// eDataMappingVarNames.peakshavebox_Powermonitor_ar_ApparentPower_L1: 				st_Variable:= IotExtractType(monitor.peakshavebox.Powermonitor.ar_ApparentPower[1], 1, 1); 
// eDataMappingVarNames.peakshavebox_Powermonitor_ar_ApparentPower_L2: 				st_Variable:= IotExtractType(monitor.peakshavebox.Powermonitor.ar_ApparentPower[2], 1, 1); 
// eDataMappingVarNames.peakshavebox_Powermonitor_ar_ApparentPower_L3: 				st_Variable:= IotExtractType(monitor.peakshavebox.Powermonitor.ar_ApparentPower[3], 1, 1); 
// eDataMappingVarNames.peakshavebox_Powermonitor_ar_ReactivePower_AVG: 				st_Variable:= IotExtractType(monitor.peakshavebox.Powermonitor.ar_ReactivePower[0], 1, 1); 
// eDataMappingVarNames.peakshavebox_Powermonitor_ar_ReactivePower_L1: 				st_Variable:= IotExtractType(monitor.peakshavebox.Powermonitor.ar_ReactivePower[1], 1, 1); 
// eDataMappingVarNames.peakshavebox_Powermonitor_ar_ReactivePower_L2: 				st_Variable:= IotExtractType(monitor.peakshavebox.Powermonitor.ar_ReactivePower[2], 1, 1); 
// eDataMappingVarNames.peakshavebox_Powermonitor_ar_ReactivePower_L3: 				st_Variable:= IotExtractType(monitor.peakshavebox.Powermonitor.ar_ReactivePower[3], 1, 1); 
// eDataMappingVarNames.peakshavebox_Powermonitor_ar_ActivePower_AVG: 				st_Variable:= IotExtractType(monitor.peakshavebox.Powermonitor.ar_ActivePower[0], 1, 1); 
// eDataMappingVarNames.peakshavebox_Powermonitor_ar_ActivePower_L1: 				st_Variable:= IotExtractType(monitor.peakshavebox.Powermonitor.ar_ActivePower[1], 1, 1); 
// eDataMappingVarNames.peakshavebox_Powermonitor_ar_ActivePower_L2: 				st_Variable:= IotExtractType(monitor.peakshavebox.Powermonitor.ar_ActivePower[2], 1, 1); 
// eDataMappingVarNames.peakshavebox_Powermonitor_ar_ActivePower_L3: 				st_Variable:= IotExtractType(monitor.peakshavebox.Powermonitor.ar_ActivePower[3], 1, 1); 
// eDataMappingVarNames.peakshavebox_Powermonitor_r_EnergyConsumed: 				st_Variable:= IotExtractType(monitor.peakshavebox.Powermonitor.r_EnergyConsumed, 0, 0); 
// eDataMappingVarNames.peakshavebox_Powermonitor_r_EnergySupplied: 				st_Variable:= IotExtractType(monitor.peakshavebox.Powermonitor.r_EnergySupplied, 0, 0); 
// eDataMappingVarNames.peakshavebox_Powermonitor_ar_THD_AVG: 				st_Variable:= IotExtractType(monitor.peakshavebox.Powermonitor.ar_THD[0], 1, 0); 
// eDataMappingVarNames.peakshavebox_Powermonitor_ar_THD_L1: 				st_Variable:= IotExtractType(monitor.peakshavebox.Powermonitor.ar_THD[1], 1, 0); 
// eDataMappingVarNames.peakshavebox_Powermonitor_ar_THD_L2: 				st_Variable:= IotExtractType(monitor.peakshavebox.Powermonitor.ar_THD[2], 1, 0); 
// eDataMappingVarNames.peakshavebox_Powermonitor_ar_THD_L3: 				st_Variable:= IotExtractType(monitor.peakshavebox.Powermonitor.ar_THD[3], 1, 0); 
// eDataMappingVarNames.peakshavebox_Powermonitor_ar_PowerFactor_AVG: 				st_Variable:= IotExtractType(monitor.peakshavebox.Powermonitor.ar_PowerFactor[0], 2, 0); 
// eDataMappingVarNames.peakshavebox_Powermonitor_ar_PowerFactor_L1: 				st_Variable:= IotExtractType(monitor.peakshavebox.Powermonitor.ar_PowerFactor[1], 2, 0); 
// eDataMappingVarNames.peakshavebox_Powermonitor_ar_PowerFactor_L2: 				st_Variable:= IotExtractType(monitor.peakshavebox.Powermonitor.ar_PowerFactor[2], 2, 0); 
// eDataMappingVarNames.peakshavebox_Powermonitor_ar_PowerFactor_L3: 				st_Variable:= IotExtractType(monitor.peakshavebox.Powermonitor.ar_PowerFactor[3], 2, 0); 
// eDataMappingVarNames.peakshavebox_Powermonitor_ar_Current_AVG: 				st_Variable:= IotExtractType(monitor.peakshavebox.Powermonitor.ar_Current[0], 1, 1); 
// eDataMappingVarNames.peakshavebox_Powermonitor_ar_Current_L1: 				st_Variable:= IotExtractType(monitor.peakshavebox.Powermonitor.ar_Current[1], 1, 1); 
// eDataMappingVarNames.peakshavebox_Powermonitor_ar_Current_L2: 				st_Variable:= IotExtractType(monitor.peakshavebox.Powermonitor.ar_Current[2], 1, 1); 
// eDataMappingVarNames.peakshavebox_Powermonitor_ar_Current_L3: 				st_Variable:= IotExtractType(monitor.peakshavebox.Powermonitor.ar_Current[3], 1, 1); 
// eDataMappingVarNames.peakshavebox_Powermonitor_ar_Current_N: 				st_Variable:= IotExtractType(monitor.peakshavebox.Powermonitor.ar_Current[4], 1, 1); 
// eDataMappingVarNames.peakshavebox_Powermonitor_r_CurrentUnbalance: 				st_Variable:= IotExtractType(monitor.peakshavebox.Powermonitor.r_CurrentUnbalance, 1, 0); 
// eDataMappingVarNames.peakshavebox_Powermonitor_e_ACrotationStatus: 				st_Variable:= IotExtractType(monitor.peakshavebox.Powermonitor.e_ACrotationStatus, 0, 0); 
// eDataMappingVarNames.peakshavebox_Powermonitor_ar_PhaseVoltage_AVG: 				st_Variable:= IotExtractType(monitor.peakshavebox.Powermonitor.ar_PhaseVoltage[0], 0, 0); 
// eDataMappingVarNames.peakshavebox_Powermonitor_ar_PhaseVoltage_L1: 				st_Variable:= IotExtractType(monitor.peakshavebox.Powermonitor.ar_PhaseVoltage[1], 1, 1); 
// eDataMappingVarNames.peakshavebox_Powermonitor_ar_PhaseVoltage_L2: 				st_Variable:= IotExtractType(monitor.peakshavebox.Powermonitor.ar_PhaseVoltage[2], 1, 1); 
// eDataMappingVarNames.peakshavebox_Powermonitor_ar_PhaseVoltage_L3: 				st_Variable:= IotExtractType(monitor.peakshavebox.Powermonitor.ar_PhaseVoltage[3], 1, 1); 
// eDataMappingVarNames.peakshavebox_Powermonitor_ar_LineVoltage_AVG: 				st_Variable:= IotExtractType(monitor.peakshavebox.Powermonitor.ar_LineVoltage[0], 1, 1); 
// eDataMappingVarNames.peakshavebox_Powermonitor_ar_LineVoltage_L1: 				st_Variable:= IotExtractType(monitor.peakshavebox.Powermonitor.ar_LineVoltage[1], 1, 1); 
// eDataMappingVarNames.peakshavebox_Powermonitor_ar_LineVoltage_L2: 				st_Variable:= IotExtractType(monitor.peakshavebox.Powermonitor.ar_LineVoltage[2], 1, 1); 
// eDataMappingVarNames.peakshavebox_Powermonitor_ar_LineVoltage_L3: 				st_Variable:= IotExtractType(monitor.peakshavebox.Powermonitor.ar_LineVoltage[3], 1, 1); 
// eDataMappingVarNames.peakshavebox_Powermonitor_li_TimeVoltZeroCrossup: 				st_Variable:= IotExtractType(monitor.peakshavebox.Powermonitor.li_TimeVoltZeroCrossup, 0, 0); 
// eDataMappingVarNames.peakshavebox_Powermonitor_ar_Frequency_AVG: 				st_Variable:= IotExtractType(monitor.peakshavebox.Powermonitor.ar_Frequency[0], 2, 1); 
// eDataMappingVarNames.peakshavebox_Powermonitor_ar_Frequency_L1: 				st_Variable:= IotExtractType(monitor.peakshavebox.Powermonitor.ar_Frequency[1], 2, 1); 
// eDataMappingVarNames.peakshavebox_Powermonitor_ar_Frequency_L2: 				st_Variable:= IotExtractType(monitor.peakshavebox.Powermonitor.ar_Frequency[2], 2, 1); 
// eDataMappingVarNames.peakshavebox_Powermonitor_ar_Frequency_L3: 				st_Variable:= IotExtractType(monitor.peakshavebox.Powermonitor.ar_Frequency[3], 2, 1); 
// eDataMappingVarNames.peakshavebox_Powermonitor_r_VoltageUnbalance: 				st_Variable:= IotExtractType(monitor.peakshavebox.Powermonitor.r_VoltageUnbalance, 1, 0); 
// eDataMappingVarNames.peakshavebox_PowerStatus_b_RotaryField: 				st_Variable:= IotExtractType(monitor.peakshavebox.PowerStatus.b_RotaryField, 0, 0); 
// eDataMappingVarNames.peakshavebox_PowerStatus_b_GeneralWarning: 				st_Variable:= IotExtractType(monitor.peakshavebox.PowerStatus.b_GeneralWarning, 0, 0); 
// eDataMappingVarNames.peakshavebox_PowerStatus_b_GeneralFault: 				st_Variable:= IotExtractType(monitor.peakshavebox.PowerStatus.b_GeneralFault, 0, 0); 
// eDataMappingVarNames.peakshavebox_PowerStatus_b_OverVoltage: 				st_Variable:= IotExtractType(monitor.peakshavebox.PowerStatus.b_OverVoltage, 0, 0); 
// eDataMappingVarNames.peakshavebox_PowerStatus_b_UnderVoltage: 				st_Variable:= IotExtractType(monitor.peakshavebox.PowerStatus.b_UnderVoltage, 0, 0); 
// eDataMappingVarNames.peakshavebox_PowerStatus_b_OverCurrent: 				st_Variable:= IotExtractType(monitor.peakshavebox.PowerStatus.b_OverCurrent, 0, 0); 
// eDataMappingVarNames.peakshavebox_PowerStatus_b_Error_Phase_1: 				st_Variable:= IotExtractType(monitor.peakshavebox.PowerStatus.b_Error_Phase[1], 0, 0); 
// eDataMappingVarNames.peakshavebox_PowerStatus_b_Error_Phase_2: 				st_Variable:= IotExtractType(monitor.peakshavebox.PowerStatus.b_Error_Phase[2], 0, 0); 
// eDataMappingVarNames.peakshavebox_PowerStatus_b_Error_Phase_3: 				st_Variable:= IotExtractType(monitor.peakshavebox.PowerStatus.b_Error_Phase[3], 0, 0); 
// eDataMappingVarNames.peakshavebox_r_MaxCTCurrent: 				st_Variable:= IotExtractType(monitor.peakshavebox.r_MaxCTCurrent, 0, 0); 
// eDataMappingVarNames.peakshavebox_b_buscouplerReady: 				st_Variable:= IotExtractType(monitor.peakshavebox.b_buscouplerReady, 0, 0); 
// eDataMappingVarNames.peakshavebox_b_active: 				st_Variable:= IotExtractType(monitor.peakshavebox.b_active, 0, 0); 
// eDataMappingVarNames.peakshavebox_b_dataOK: 				st_Variable:= IotExtractType(monitor.peakshavebox.b_dataOK, 0, 0); 
// eDataMappingVarNames.peakshavebox_b_ContactorFb: 				st_Variable:= IotExtractType(monitor.peakshavebox.b_ContactorFb, 0, 0); 
// eDataMappingVarNames.peakshavebox_b_SyncFb: 				st_Variable:= IotExtractType(monitor.peakshavebox.b_SyncFb, 0, 0); 
// eDataMappingVarNames.peakshavebox_b_SettingsChangePending: 				st_Variable:= IotExtractType(monitor.peakshavebox.b_SettingsChangePending, 0, 0); 
// eDataMappingVarNames.enclosure_climate_r_Humidity: 				st_Variable:= IotExtractType(monitor.enclosure.climate.r_Humidity, 1, 0); 
// eDataMappingVarNames.enclosure_climate_r_Temperature: 				st_Variable:= IotExtractType(monitor.enclosure.climate.r_Temperature, 1, 0); 
// eDataMappingVarNames.enclosure_climate_events_b_HumidityHigh: 				st_Variable:= IotExtractType(monitor.enclosure.climate.events.b_HumidityHigh, 0, 0); 
// eDataMappingVarNames.enclosure_climate_events_b_HumidityTooHigh: 				st_Variable:= IotExtractType(monitor.enclosure.climate.events.b_HumidityTooHigh, 0, 0); 
// eDataMappingVarNames.enclosure_climate_events_b_TemperatureHigh: 				st_Variable:= IotExtractType(monitor.enclosure.climate.events.b_TemperatureHigh, 0, 0); 
// eDataMappingVarNames.enclosure_climate_events_b_TemperatureTooHigh: 				st_Variable:= IotExtractType(monitor.enclosure.climate.events.b_TemperatureTooHigh, 0, 0); 
// eDataMappingVarNames.enclosure_climate_events_b_TemperatureLow: 				st_Variable:= IotExtractType(monitor.enclosure.climate.events.b_TemperatureLow, 0, 0); 
// eDataMappingVarNames.enclosure_climate_events_b_TemperatureTooLow: 				st_Variable:= IotExtractType(monitor.enclosure.climate.events.b_TemperatureTooLow, 0, 0); 
// eDataMappingVarNames.enclosure_climate_events_b_AIOverrange: 				st_Variable:= IotExtractType(monitor.enclosure.climate.events.b_AIOverrange, 0, 0); 
// eDataMappingVarNames.enclosure_climate_events_b_AIUnderrange: 				st_Variable:= IotExtractType(monitor.enclosure.climate.events.b_AIUnderrange, 0, 0); 
// eDataMappingVarNames.enclosure_climate_events_b_AIError: 				st_Variable:= IotExtractType(monitor.enclosure.climate.events.b_AIError, 0, 0); 
// eDataMappingVarNames.enclosure_climate_events_b_DewpointTooHigh: 				st_Variable:= IotExtractType(monitor.enclosure.climate.events.b_DewpointTooHigh, 0, 0); 
// //eDataMappingVarNames.enclosure_doors_b_ClientpanelDoorClosed: 				st_Variable:= IotExtractType(monitor.enclosure.doors.b_ClientpanelDoorClosed, 0, 0); 
// //eDataMappingVarNames.enclosure_doors_b_ControlPanelDoorClosed: 				st_Variable:= IotExtractType(monitor.enclosure.doors.b_ControlPanelDoorClosed, 0, 0); 
// eDataMappingVarNames.enclosure_ledstrip_b_error: 				st_Variable:= IotExtractType(monitor.enclosure.ledstrip.b_error, 0, 0); 
// eDataMappingVarNames.enclosure_ledstrip_BeckhoffLed: 				st_Variable:= IotExtractType(monitor.enclosure.ledstrip.BeckhoffLed, 0, 0); 
// eDataMappingVarNames.internalpsu_b_24VdcAvailable: 				st_Variable:= IotExtractType(monitor.internalpsu.b_24VdcAvailable, 0, 0); 
// eDataMappingVarNames.internalpsu_b_HVDCAvailable: 				st_Variable:= IotExtractType(monitor.internalpsu.b_HVDCAvailable, 0, 0); 
// eDataMappingVarNames.internalpsu_b_400VACAvailable: 				st_Variable:= IotExtractType(monitor.internalpsu.b_400VACAvailable, 0, 0); 
// //eDataMappingVarNames.internalpsu_e_400VSupplySource: 				st_Variable:= IotExtractType(monitor.internalpsu.e_400VSupplySource, 0, 0); 
// eDataMappingVarNames.internalpsu_UPS_r_InputVoltage: 				st_Variable:= IotExtractType(monitor.internalpsu.UPS.r_InputVoltage, 1, 1); 
// eDataMappingVarNames.internalpsu_UPS_r_OutputVoltage: 				st_Variable:= IotExtractType(monitor.internalpsu.UPS.r_OutputVoltage, 1, 1); 
// eDataMappingVarNames.internalpsu_UPS_r_BatteryVoltage: 				st_Variable:= IotExtractType(monitor.internalpsu.UPS.r_BatteryVoltage, 1, 1); 
// eDataMappingVarNames.internalpsu_UPS_r_OutputCurrent: 				st_Variable:= IotExtractType(monitor.internalpsu.UPS.r_OutputCurrent, 2, 0); 
// eDataMappingVarNames.internalpsu_UPS_ui_SOC: 				st_Variable:= IotExtractType(monitor.internalpsu.UPS.ui_SOC, 0, 0); 
// eDataMappingVarNames.internalpsu_UPS_b_ChargerActive: 				st_Variable:= IotExtractType(monitor.internalpsu.UPS.b_ChargerActive, 0, 0); 
// eDataMappingVarNames.internalpsu_UPS_b_SystemOnBattery: 				st_Variable:= IotExtractType(monitor.internalpsu.UPS.b_SystemOnBattery, 0, 0); 
// eDataMappingVarNames.internalpsu_UPS_b_SystemOnDCInput: 				st_Variable:= IotExtractType(monitor.internalpsu.UPS.b_SystemOnDCInput, 0, 0); 
// eDataMappingVarNames.internalpsu_UPS_Events_b_BatteryLowInfo: 				st_Variable:= IotExtractType(monitor.internalpsu.UPS.Events.b_BatteryLowInfo, 0, 0); 
// eDataMappingVarNames.internalpsu_UPS_Events_b_BatteryLowWarning: 				st_Variable:= IotExtractType(monitor.internalpsu.UPS.Events.b_BatteryLowWarning, 0, 0); 
// eDataMappingVarNames.internalpsu_UPS_Events_b_BatteryLowError: 				st_Variable:= IotExtractType(monitor.internalpsu.UPS.Events.b_BatteryLowError, 0, 0); 
// eDataMappingVarNames.internalpsu_UPS_Events_b_NoBatteryError: 				st_Variable:= IotExtractType(monitor.internalpsu.UPS.Events.b_NoBatteryError, 0, 0); 
// eDataMappingVarNames.internalpsu_UPS_Events_b_InputVoltageWarning: 				st_Variable:= IotExtractType(monitor.internalpsu.UPS.Events.b_InputVoltageWarning, 0, 0); 
// eDataMappingVarNames.internalpsu_Events_b_DCPSUFault: 				st_Variable:= IotExtractType(monitor.internalpsu.Events.b_DCPSUFault, 0, 0); 
// eDataMappingVarNames.internalpsu_Events_b_ACPSUFault: 				st_Variable:= IotExtractType(monitor.internalpsu.Events.b_ACPSUFault, 0, 0); 
// eDataMappingVarNames.internalpsu_Events_b_GridInputFuseTripped: 				st_Variable:= IotExtractType(monitor.internalpsu.Events.b_GridInputFuseTripped, 0, 0); 
// //eDataMappingVarNames.internalpsu_Events_b_CEEInputFuseTripped: 				st_Variable:= IotExtractType(monitor.internalpsu.Events.b_CEEInputFuseTripped, 0, 0); 
// eDataMappingVarNames.internalpsu_Events_b_HVDCShutdownTimeExceeded: 				st_Variable:= IotExtractType(monitor.internalpsu.Events.b_HVDCShutdownTimeExceeded, 0, 0); 
// eDataMappingVarNames.internalpsu_Events_b_UPSLowShutdown: 				st_Variable:= IotExtractType(monitor.internalpsu.Events.b_UPSLowShutdown, 0, 0); 
// eDataMappingVarNames.PLC_r_CPUload: 				st_Variable:= IotExtractType(monitor.PLC.r_CPUload, 0, 0); 
// eDataMappingVarNames.PLC_e_ProfinetState: 				st_Variable:= IotExtractType(monitor.PLC.e_ProfinetState, 0, 0); 
// eDataMappingVarNames.PLC_e_EthercatState: 				st_Variable:= IotExtractType(monitor.PLC.e_EthercatState, 0, 0); 
// eDataMappingVarNames.Cooling_CoolingSystemMode: 				st_Variable:= IotExtractType(monitor.Cooling.CoolingSystemMode, 0, 0); 
// eDataMappingVarNames.Cooling_HeatPumpStatus: 				st_Variable:= IotExtractType(monitor.Cooling.HeatPumpStatus, 0, 0); 
// eDataMappingVarNames.Cooling_r_CoolantTemperature: 				st_Variable:= IotExtractType(monitor.Cooling.r_CoolantTemperature, 1, 0); 
// eDataMappingVarNames.Cooling_r_CoolantPressure: 				st_Variable:= IotExtractType(monitor.Cooling.r_CoolantPressure, 2, 0); 
// eDataMappingVarNames.Cooling_r_EnclosureDewpoint: 				st_Variable:= IotExtractType(monitor.Cooling.r_EnclosureDewpoint, 0, 0); 
// eDataMappingVarNames.Cooling_ui_DehumRemainingTime: 				st_Variable:= IotExtractType(monitor.Cooling.ui_DehumRemainingTime, 0, 0); 
// eDataMappingVarNames.Cooling_HeatPumpSystem_HeatPumpStatus: 				st_Variable:= IotExtractType(monitor.Cooling.HeatPumpStatus, 0, 0); 
// eDataMappingVarNames.Cooling_HeatPumpSystem_PrimaryHeatpumpGet_HeatPumpState: 				st_Variable:= IotExtractType(monitor.Cooling.HeatPumpStatus, 0, 0); {warning 'needs revision, heatpump now doesn't have individuals state'} 
// eDataMappingVarNames.Cooling_HeatPumpSystem_PrimaryHeatpumpGet_Setpoint: 				st_Variable:= IotExtractType(monitor.Cooling.Heatpump.Setpoint, 0, 0); 
// eDataMappingVarNames.Cooling_HeatPumpSystem_PrimaryHeatpumpGet_Events_b_CommWarning: 				st_Variable:= IotExtractType(monitor.Cooling.Heatpump.Events.b_CommWarning, 0, 0); 
// eDataMappingVarNames.Cooling_HeatPumpSystem_PrimaryHeatpumpGet_Events_b_ProbeError: 				st_Variable:= IotExtractType(monitor.Cooling.Heatpump.Events.b_ProbeError, 0, 0); 
// eDataMappingVarNames.Cooling_HeatPumpSystem_PrimaryHeatpumpGet_Events_b_PressureError: 				st_Variable:= IotExtractType(monitor.Cooling.Heatpump.Events.b_PressureError, 0, 0); 
// eDataMappingVarNames.Cooling_HeatPumpSystem_PrimaryHeatpumpGet_Events_b_CompressorError: 				st_Variable:= IotExtractType(monitor.Cooling.Heatpump.Events.b_CompressorError, 0, 0); 
// eDataMappingVarNames.Cooling_HeatPumpSystem_PrimaryHeatpumpGet_Events_b_ValveError: 				st_Variable:= IotExtractType(monitor.Cooling.Heatpump.Events.b_ValveError, 0, 0); 
// eDataMappingVarNames.Cooling_HeatPumpSystem_PrimaryHeatpumpGet_Events_b_FanError: 				st_Variable:= IotExtractType(monitor.Cooling.Heatpump.Events.b_FanError, 0, 0); 
// eDataMappingVarNames.Cooling_HeatPumpSystem_PrimaryHeatpumpGet_Events_b_PumpError: 				st_Variable:= IotExtractType(monitor.Cooling.Heatpump.Events.b_PumpError, 0, 0); 
// eDataMappingVarNames.Cooling_HeatPumpSystem_PrimaryHeatpumpGet_Events_b_WaterTempError: 				st_Variable:= IotExtractType(monitor.Cooling.Heatpump.Events.b_WaterTempError, 0, 0); 
// eDataMappingVarNames.Cooling_HeatPumpSystem_PrimaryHeatpumpGet_Events_b_IOError: 				st_Variable:= IotExtractType(monitor.Cooling.Heatpump.Events.b_IOError, 0, 0); 
// eDataMappingVarNames.Cooling_HeatPumpSystem_PrimaryHeatpumpGet_Events_b_HeatpumpPreheatingActive: 				st_Variable:= IotExtractType(monitor.Cooling.Heatpump.Events.b_HeatpumpPreheatingActive, 0, 0); 
// eDataMappingVarNames.Cooling_HeatPumpSystem_PrimaryHeatpumpGet_Events_b_TooColdForHeatpumpHeating: 				st_Variable:= IotExtractType(monitor.Cooling.Heatpump.Events.b_TooColdForHeatpumpHeating, 0, 0); 
// eDataMappingVarNames.Cooling_HeatPumpSystem_PrimaryHeatpumpGet_HeatpumpData_i_FW_Version: 				st_Variable:= IotExtractType(monitor.Cooling.Heatpump.HeatpumpData.i_FW_Version, 0, 0); 
// eDataMappingVarNames.Cooling_HeatPumpSystem_PrimaryHeatpumpGet_HeatpumpData_i_FW_release: 				st_Variable:= IotExtractType(monitor.Cooling.Heatpump.HeatpumpData.i_FW_release, 0, 0); 
// eDataMappingVarNames.Cooling_HeatPumpSystem_PrimaryHeatpumpGet_HeatpumpData_w_FW_Subrelease: 				st_Variable:= IotExtractType(monitor.Cooling.Heatpump.HeatpumpData.HeatpumpData.w_FW_Subrelease, 0, 0); 
// eDataMappingVarNames.Cooling_HeatPumpSystem_PrimaryHeatpumpGet_HeatpumpData_w_FW_creationDate: 				st_Variable:= IotExtractType(monitor.Cooling.Heatpump.Heatpumpdata.w_FW_creationDate, 0, 0); 
// eDataMappingVarNames.Cooling_HeatPumpSystem_PrimaryHeatpumpGet_HeatpumpData_w_Serialnumber_0: 				st_Variable:= IotExtractType(monitor.Cooling.Heatpump.Heatpumpdata.w_Serialnumber[0], 0, 0); 
// eDataMappingVarNames.Cooling_HeatPumpSystem_PrimaryHeatpumpGet_HeatpumpData_w_Serialnumber_1: 				st_Variable:= IotExtractType(monitor.Cooling.Heatpump.Heatpumpdata.w_Serialnumber[1], 0, 0); 
// eDataMappingVarNames.Cooling_HeatPumpSystem_PrimaryHeatpumpGet_HeatpumpData_w_Serialnumber_2: 				st_Variable:= IotExtractType(monitor.Cooling.Heatpump.Heatpumpdata.w_Serialnumber[2], 0, 0); 
// eDataMappingVarNames.Cooling_HeatPumpSystem_PrimaryHeatpumpGet_HeatpumpData_w_Serialnumber_3: 				st_Variable:= IotExtractType(monitor.Cooling.Heatpump.Heatpumpdata.w_Serialnumber[3], 0, 0); 
// eDataMappingVarNames.Cooling_HeatPumpSystem_PrimaryHeatpumpGet_HeatpumpData_w_Serialnumber_4: 				st_Variable:= IotExtractType(monitor.Cooling.Heatpump.Heatpumpdata.w_Serialnumber[4], 0, 0); 
// eDataMappingVarNames.Cooling_HeatPumpSystem_PrimaryHeatpumpGet_HeatpumpData_w_Serialnumber_5: 				st_Variable:= IotExtractType(monitor.Cooling.Heatpump.Heatpumpdata.w_Serialnumber[5], 0, 0); 
// eDataMappingVarNames.Cooling_HeatPumpSystem_PrimaryHeatpumpGet_HeatpumpData_w_Serialnumber_6: 				st_Variable:= IotExtractType(monitor.Cooling.Heatpump.Heatpumpdata.w_Serialnumber[6], 0, 0); 
// eDataMappingVarNames.Cooling_HeatPumpSystem_PrimaryHeatpumpGet_HeatpumpData_w_Serialnumber_7: 				st_Variable:= IotExtractType(monitor.Cooling.Heatpump.Heatpumpdata.w_Serialnumber[7], 0, 0); 
// eDataMappingVarNames.Cooling_HeatPumpSystem_PrimaryHeatpumpGet_HeatpumpData_w_Serialnumber_8: 				st_Variable:= IotExtractType(monitor.Cooling.Heatpump.Heatpumpdata.w_Serialnumber[8], 0, 0); 
// eDataMappingVarNames.Cooling_HeatPumpSystem_PrimaryHeatpumpGet_HeatpumpData_w_Serialnumber_9: 				st_Variable:= IotExtractType(monitor.Cooling.Heatpump.Heatpumpdata.w_Serialnumber[9], 0, 0); 
// eDataMappingVarNames.Cooling_HeatPumpSystem_PrimaryHeatpumpGet_HeatpumpData_w_Serialnumber_10: 				st_Variable:= IotExtractType(monitor.Cooling.Heatpump.Heatpumpdata.w_Serialnumber[10], 0, 0); 
// eDataMappingVarNames.Cooling_HeatPumpSystem_PrimaryHeatpumpGet_HeatpumpData_w_Serialnumber_11: 				st_Variable:= IotExtractType(monitor.Cooling.Heatpump.Heatpumpdata.w_Serialnumber[11], 0, 0); 
// eDataMappingVarNames.Cooling_HeatPumpSystem_PrimaryHeatpumpGet_HeatpumpData_w_Serialnumber_12: 				st_Variable:= IotExtractType(monitor.Cooling.Heatpump.Heatpumpdata.w_Serialnumber[12], 0, 0); 
// eDataMappingVarNames.Cooling_HeatPumpSystem_PrimaryHeatpumpGet_HeatpumpData_w_Serialnumber_13: 				st_Variable:= IotExtractType(monitor.Cooling.Heatpump.Heatpumpdata.w_Serialnumber[13], 0, 0); 
// eDataMappingVarNames.Cooling_HeatPumpSystem_PrimaryHeatpumpGet_HeatpumpData_w_Serialnumber_14: 				st_Variable:= IotExtractType(monitor.Cooling.Heatpump.Heatpumpdata.w_Serialnumber[14], 0, 0); 
// eDataMappingVarNames.Cooling_HeatPumpSystem_PrimaryHeatpumpGet_HeatpumpData_w_Serialnumber_15: 				st_Variable:= IotExtractType(monitor.Cooling.Heatpump.Heatpumpdata.w_Serialnumber[15], 0, 0); 
// eDataMappingVarNames.Cooling_HeatPumpSystem_PrimaryHeatpumpGet_HeatpumpData_w_Serialnumber_16: 				st_Variable:= IotExtractType(monitor.Cooling.Heatpump.Heatpumpdata.w_Serialnumber[16], 0, 0); 
// eDataMappingVarNames.Cooling_HeatPumpSystem_PrimaryHeatpumpGet_HeatpumpData_w_Serialnumber_17: 				st_Variable:= IotExtractType(monitor.Cooling.Heatpump.Heatpumpdata.w_Serialnumber[17], 0, 0); 
// eDataMappingVarNames.Cooling_HeatPumpSystem_PrimaryHeatpumpGet_HeatpumpData_i_OperatingHours: 				st_Variable:= IotExtractType(monitor.Cooling.Heatpump.Heatpumpdata.i_OperatingHours, 0, 0); 
// eDataMappingVarNames.Cooling_HeatPumpSystem_PrimaryHeatpumpGet_HeatpumpData_r_CoolantPower: 				st_Variable:= IotExtractType(monitor.Cooling.Heatpump.Heatpumpdata.r_CoolantPower, 0, 0); 
// eDataMappingVarNames.Cooling_HeatPumpSystem_PrimaryHeatpumpGet_HeatpumpData_r_InletWaterTemp: 				st_Variable:= IotExtractType(monitor.Cooling.Heatpump.Heatpumpdata.r_InletWaterTemp, 0, 0); 
// eDataMappingVarNames.Cooling_HeatPumpSystem_PrimaryHeatpumpGet_HeatpumpData_r_OutletWaterTemp: 				st_Variable:= IotExtractType(monitor.Cooling.Heatpump.Heatpumpdata.r_OutletWaterTemp, 0, 0); 
// eDataMappingVarNames.Cooling_HeatPumpSystem_PrimaryHeatpumpGet_HeatpumpData_r_HighPressure: 				st_Variable:= IotExtractType(monitor.Cooling.Heatpump.Heatpumpdata.r_HighPressure, 0, 0); 
// eDataMappingVarNames.Cooling_HeatPumpSystem_PrimaryHeatpumpGet_HeatpumpData_r_LowPressure: 				st_Variable:= IotExtractType(monitor.Cooling.HeatPump.HeatpumpData.r_LowPressure, 0, 0); 
// eDataMappingVarNames.Cooling_HeatPumpSystem_PrimaryHeatpumpGet_HeatpumpData_r_CompInputTemp: 				st_Variable:= IotExtractType(monitor.Cooling.Heatpump.HeatpumpData.r_CompInputTemp, 0, 0); 
// eDataMappingVarNames.Cooling_HeatPumpSystem_PrimaryHeatpumpGet_HeatpumpData_r_OutdoorTemp: 				st_Variable:= IotExtractType(monitor.Cooling.Heatpump.HeatpumpData.r_OutdoorTemp, 0, 0); 
// eDataMappingVarNames.Cooling_HeatPumpSystem_PrimaryHeatpumpGet_HeatpumpData_r_CompOutputTemp: 				st_Variable:= IotExtractType(monitor.Cooling.Heatpump.HeatpumpData.r_CompOutputTemp, 0, 0); 
// eDataMappingVarNames.Cooling_HeatPumpSystem_PrimaryHeatpumpGet_HeatpumpData_ui_WaterFlowRate: 				st_Variable:= IotExtractType(monitor.Cooling.Heatpump.HeatpumpData.ui_WaterFlowRate, 0, 0); 
// eDataMappingVarNames.Cooling_HeatPumpSystem_PrimaryHeatpumpGet_HeatpumpData_w_ErrorList_1: 				st_Variable:= IotExtractType(monitor.Cooling.Heatpump.HeatpumpData.w_ErrorList[1], 0, 0); 
// eDataMappingVarNames.Cooling_HeatPumpSystem_PrimaryHeatpumpGet_HeatpumpData_w_ErrorList_2: 				st_Variable:= IotExtractType(monitor.Cooling.Heatpump.HeatpumpData.w_ErrorList[2], 0, 0); 
// eDataMappingVarNames.Cooling_HeatPumpSystem_PrimaryHeatpumpGet_HeatpumpData_w_ErrorList_3: 				st_Variable:= IotExtractType(monitor.Cooling.Heatpump.HeatpumpData.w_ErrorList[3], 0, 0); 
// eDataMappingVarNames.Cooling_HeatPumpSystem_PrimaryHeatpumpGet_HeatpumpData_w_ErrorList_4: 				st_Variable:= IotExtractType(monitor.Cooling.Heatpump.HeatpumpData.w_ErrorList[4], 0, 0); 
// eDataMappingVarNames.Cooling_HeatPumpSystem_PrimaryHeatpumpGet_HeatpumpData_w_ErrorList_5: 				st_Variable:= IotExtractType(monitor.Cooling.Heatpump.HeatpumpData.w_ErrorList[5], 0, 0); 
// eDataMappingVarNames.Cooling_HeatPumpSystem_PrimaryHeatpumpGet_HeatpumpData_w_ErrorList_6: 				st_Variable:= IotExtractType(monitor.Cooling.Heatpump.HeatpumpData.w_ErrorList[6], 0, 0); 
// eDataMappingVarNames.Cooling_HeatPumpSystem_PrimaryHeatpumpGet_HeatpumpData_w_ErrorList_7: 				st_Variable:= IotExtractType(monitor.Cooling.Heatpump.HeatpumpData.w_ErrorList[7], 0, 0); 
// eDataMappingVarNames.Cooling_HeatPumpSystem_PrimaryHeatpumpGet_HeatpumpData_r_FanSpeedPCT: 				st_Variable:= IotExtractType(monitor.Cooling.Heatpump.HeatpumpData.r_FanSpeedPCT, 0, 0); 
// eDataMappingVarNames.Cooling_HeatPumpSystem_PrimaryHeatpumpGet_HeatpumpData_r_PumpSpeedPCT: 				st_Variable:= IotExtractType(monitor.Cooling.Heatpump.HeatpumpData.r_PumpSpeedPCT, 0, 0); 
// eDataMappingVarNames.Cooling_HeatPumpSystem_PrimaryHeatpumpGet_HeatpumpData_r_SetpointHeating: 				st_Variable:= IotExtractType(monitor.Cooling.Heatpump.HeatpumpData.r_SetpointHeating, 1, 0); 
// eDataMappingVarNames.Cooling_HeatPumpSystem_PrimaryHeatpumpGet_HeatpumpData_r_SetpointCooling: 				st_Variable:= IotExtractType(monitor.Cooling.Heatpump.HeatpumpData.r_SetpointCooling, 1, 0); 
// eDataMappingVarNames.Cooling_HeatPumpSystem_PrimaryHeatpumpGet_HeatpumpData_b_DefrostingActive: 				st_Variable:= IotExtractType(monitor.Cooling.Heatpump.HeatpumpData.b_DefrostingActive, 0, 0); 
// eDataMappingVarNames.Cooling_HeatPumpSystem_SecondaryHeatpumpGet_HeatPumpState: 				st_Variable:= IotExtractType(monitor.Cooling.HeatPumpSystem.SecondaryHeatpumpGet.HeatPumpState, 0, 0); 
// eDataMappingVarNames.Cooling_HeatPumpSystem_SecondaryHeatpumpGet_Setpoint: 				st_Variable:= IotExtractType(monitor.Cooling.HeatPumpSystem.SecondaryHeatpumpGet.Setpoint, 0, 0); 
// eDataMappingVarNames.Cooling_HeatPumpSystem_SecondaryHeatpumpGet_Events_b_CommWarning: 				st_Variable:= IotExtractType(monitor.Cooling.HeatPumpSystem.SecondaryHeatpumpGet.Events.b_CommWarning, 0, 0); 
// eDataMappingVarNames.Cooling_HeatPumpSystem_SecondaryHeatpumpGet_Events_b_ProbeError: 				st_Variable:= IotExtractType(monitor.Cooling.HeatPumpSystem.SecondaryHeatpumpGet.Events.b_ProbeError, 0, 0); 
// eDataMappingVarNames.Cooling_HeatPumpSystem_SecondaryHeatpumpGet_Events_b_PressureError: 				st_Variable:= IotExtractType(monitor.Cooling.HeatPumpSystem.SecondaryHeatpumpGet.Events.b_PressureError, 0, 0); 
// eDataMappingVarNames.Cooling_HeatPumpSystem_SecondaryHeatpumpGet_Events_b_CompressorError: 				st_Variable:= IotExtractType(monitor.Cooling.HeatPumpSystem.SecondaryHeatpumpGet.Events.b_CompressorError, 0, 0); 
// eDataMappingVarNames.Cooling_HeatPumpSystem_SecondaryHeatpumpGet_Events_b_ValveError: 				st_Variable:= IotExtractType(monitor.Cooling.HeatPumpSystem.SecondaryHeatpumpGet.Events.b_ValveError, 0, 0); 
// eDataMappingVarNames.Cooling_HeatPumpSystem_SecondaryHeatpumpGet_Events_b_FanError: 				st_Variable:= IotExtractType(monitor.Cooling.HeatPumpSystem.SecondaryHeatpumpGet.Events.b_FanError, 0, 0); 
// eDataMappingVarNames.Cooling_HeatPumpSystem_SecondaryHeatpumpGet_Events_b_PumpError: 				st_Variable:= IotExtractType(monitor.Cooling.HeatPumpSystem.SecondaryHeatpumpGet.Events.b_PumpError, 0, 0); 
// eDataMappingVarNames.Cooling_HeatPumpSystem_SecondaryHeatpumpGet_Events_b_WaterTempError: 				st_Variable:= IotExtractType(monitor.Cooling.HeatPumpSystem.SecondaryHeatpumpGet.Events.b_WaterTempError, 0, 0); 
// eDataMappingVarNames.Cooling_HeatPumpSystem_SecondaryHeatpumpGet_Events_b_IOError: 				st_Variable:= IotExtractType(monitor.Cooling.HeatPumpSystem.SecondaryHeatpumpGet.Events.b_IOError, 0, 0); 
// eDataMappingVarNames.Cooling_HeatPumpSystem_SecondaryHeatpumpGet_Events_b_HeatpumpPreheatingActive: 				st_Variable:= IotExtractType(monitor.Cooling.HeatPumpSystem.SecondaryHeatpumpGet.Events.b_HeatpumpPreheatingActive, 0, 0); 
// eDataMappingVarNames.Cooling_HeatPumpSystem_SecondaryHeatpumpGet_Events_b_TooColdForHeatpumpHeating: 				st_Variable:= IotExtractType(monitor.Cooling.HeatPumpSystem.SecondaryHeatpumpGet.Events.b_TooColdForHeatpumpHeating, 0, 0); 
// eDataMappingVarNames.Cooling_HeatPumpSystem_SecondaryHeatpumpGet_HeatpumpData_i_FW_Version: 				st_Variable:= IotExtractType(monitor.Cooling.HeatPumpSystem.SecondaryHeatpumpGet.HeatpumpData.i_FW_Version, 0, 0); 
// eDataMappingVarNames.Cooling_HeatPumpSystem_SecondaryHeatpumpGet_HeatpumpData_i_FW_release: 				st_Variable:= IotExtractType(monitor.Cooling.HeatPumpSystem.SecondaryHeatpumpGet.HeatpumpData.i_FW_release, 0, 0); 
// eDataMappingVarNames.Cooling_HeatPumpSystem_SecondaryHeatpumpGet_HeatpumpData_w_FW_Subrelease: 				st_Variable:= IotExtractType(monitor.Cooling.HeatPumpSystem.SecondaryHeatpumpGet.HeatpumpData.w_FW_Subrelease, 0, 0); 
// eDataMappingVarNames.Cooling_HeatPumpSystem_SecondaryHeatpumpGet_HeatpumpData_w_FW_creationDate: 				st_Variable:= IotExtractType(monitor.Cooling.HeatPumpSystem.SecondaryHeatpumpGet.HeatpumpData.w_FW_creationDate, 0, 0); 
// eDataMappingVarNames.Cooling_HeatPumpSystem_SecondaryHeatpumpGet_HeatpumpData_w_Serialnumber_0: 				st_Variable:= IotExtractType(monitor.Cooling.HeatPumpSystem.SecondaryHeatpumpGet.HeatpumpData.w_Serialnumber[0], 0, 0); 
// eDataMappingVarNames.Cooling_HeatPumpSystem_SecondaryHeatpumpGet_HeatpumpData_w_Serialnumber_1: 				st_Variable:= IotExtractType(monitor.Cooling.HeatPumpSystem.SecondaryHeatpumpGet.HeatpumpData.w_Serialnumber[1], 0, 0); 
// eDataMappingVarNames.Cooling_HeatPumpSystem_SecondaryHeatpumpGet_HeatpumpData_w_Serialnumber_2: 				st_Variable:= IotExtractType(monitor.Cooling.HeatPumpSystem.SecondaryHeatpumpGet.HeatpumpData.w_Serialnumber[2], 0, 0); 
// eDataMappingVarNames.Cooling_HeatPumpSystem_SecondaryHeatpumpGet_HeatpumpData_w_Serialnumber_3: 				st_Variable:= IotExtractType(monitor.Cooling.HeatPumpSystem.SecondaryHeatpumpGet.HeatpumpData.w_Serialnumber[3], 0, 0); 
// eDataMappingVarNames.Cooling_HeatPumpSystem_SecondaryHeatpumpGet_HeatpumpData_w_Serialnumber_4: 				st_Variable:= IotExtractType(monitor.Cooling.HeatPumpSystem.SecondaryHeatpumpGet.HeatpumpData.w_Serialnumber[4], 0, 0); 
// eDataMappingVarNames.Cooling_HeatPumpSystem_SecondaryHeatpumpGet_HeatpumpData_w_Serialnumber_5: 				st_Variable:= IotExtractType(monitor.Cooling.HeatPumpSystem.SecondaryHeatpumpGet.HeatpumpData.w_Serialnumber[5], 0, 0); 
// eDataMappingVarNames.Cooling_HeatPumpSystem_SecondaryHeatpumpGet_HeatpumpData_w_Serialnumber_6: 				st_Variable:= IotExtractType(monitor.Cooling.HeatPumpSystem.SecondaryHeatpumpGet.HeatpumpData.w_Serialnumber[6], 0, 0); 
// eDataMappingVarNames.Cooling_HeatPumpSystem_SecondaryHeatpumpGet_HeatpumpData_w_Serialnumber_7: 				st_Variable:= IotExtractType(monitor.Cooling.HeatPumpSystem.SecondaryHeatpumpGet.HeatpumpData.w_Serialnumber[7], 0, 0); 
// eDataMappingVarNames.Cooling_HeatPumpSystem_SecondaryHeatpumpGet_HeatpumpData_w_Serialnumber_8: 				st_Variable:= IotExtractType(monitor.Cooling.HeatPumpSystem.SecondaryHeatpumpGet.HeatpumpData.w_Serialnumber[8], 0, 0); 
// eDataMappingVarNames.Cooling_HeatPumpSystem_SecondaryHeatpumpGet_HeatpumpData_w_Serialnumber_9: 				st_Variable:= IotExtractType(monitor.Cooling.HeatPumpSystem.SecondaryHeatpumpGet.HeatpumpData.w_Serialnumber[9], 0, 0); 
// eDataMappingVarNames.Cooling_HeatPumpSystem_SecondaryHeatpumpGet_HeatpumpData_w_Serialnumber_10: 				st_Variable:= IotExtractType(monitor.Cooling.HeatPumpSystem.SecondaryHeatpumpGet.HeatpumpData.w_Serialnumber[10], 0, 0); 
// eDataMappingVarNames.Cooling_HeatPumpSystem_SecondaryHeatpumpGet_HeatpumpData_w_Serialnumber_11: 				st_Variable:= IotExtractType(monitor.Cooling.HeatPumpSystem.SecondaryHeatpumpGet.HeatpumpData.w_Serialnumber[11], 0, 0); 
// eDataMappingVarNames.Cooling_HeatPumpSystem_SecondaryHeatpumpGet_HeatpumpData_w_Serialnumber_12: 				st_Variable:= IotExtractType(monitor.Cooling.HeatPumpSystem.SecondaryHeatpumpGet.HeatpumpData.w_Serialnumber[12], 0, 0); 
// eDataMappingVarNames.Cooling_HeatPumpSystem_SecondaryHeatpumpGet_HeatpumpData_w_Serialnumber_13: 				st_Variable:= IotExtractType(monitor.Cooling.HeatPumpSystem.SecondaryHeatpumpGet.HeatpumpData.w_Serialnumber[13], 0, 0); 
// eDataMappingVarNames.Cooling_HeatPumpSystem_SecondaryHeatpumpGet_HeatpumpData_w_Serialnumber_14: 				st_Variable:= IotExtractType(monitor.Cooling.HeatPumpSystem.SecondaryHeatpumpGet.HeatpumpData.w_Serialnumber[14], 0, 0); 
// eDataMappingVarNames.Cooling_HeatPumpSystem_SecondaryHeatpumpGet_HeatpumpData_w_Serialnumber_15: 				st_Variable:= IotExtractType(monitor.Cooling.HeatPumpSystem.SecondaryHeatpumpGet.HeatpumpData.w_Serialnumber[15], 0, 0); 
// eDataMappingVarNames.Cooling_HeatPumpSystem_SecondaryHeatpumpGet_HeatpumpData_w_Serialnumber_16: 				st_Variable:= IotExtractType(monitor.Cooling.HeatPumpSystem.SecondaryHeatpumpGet.HeatpumpData.w_Serialnumber[16], 0, 0); 
// eDataMappingVarNames.Cooling_HeatPumpSystem_SecondaryHeatpumpGet_HeatpumpData_w_Serialnumber_17: 				st_Variable:= IotExtractType(monitor.Cooling.HeatPumpSystem.SecondaryHeatpumpGet.HeatpumpData.w_Serialnumber[17], 0, 0); 
// eDataMappingVarNames.Cooling_HeatPumpSystem_SecondaryHeatpumpGet_HeatpumpData_i_OperatingHours: 				st_Variable:= IotExtractType(monitor.Cooling.HeatPumpSystem.SecondaryHeatpumpGet.HeatpumpData.i_OperatingHours, 0, 0); 
// eDataMappingVarNames.Cooling_HeatPumpSystem_SecondaryHeatpumpGet_HeatpumpData_r_CoolantPower: 				st_Variable:= IotExtractType(monitor.Cooling.HeatPumpSystem.SecondaryHeatpumpGet.HeatpumpData.r_CoolantPower, 1, 0); 
// eDataMappingVarNames.Cooling_HeatPumpSystem_SecondaryHeatpumpGet_HeatpumpData_r_InletWaterTemp: 				st_Variable:= IotExtractType(monitor.Cooling.HeatPumpSystem.SecondaryHeatpumpGet.HeatpumpData.r_InletWaterTemp, 1, 0); 
// eDataMappingVarNames.Cooling_HeatPumpSystem_SecondaryHeatpumpGet_HeatpumpData_r_OutletWaterTemp: 				st_Variable:= IotExtractType(monitor.Cooling.HeatPumpSystem.SecondaryHeatpumpGet.HeatpumpData.r_OutletWaterTemp, 1, 0); 
// eDataMappingVarNames.Cooling_HeatPumpSystem_SecondaryHeatpumpGet_HeatpumpData_r_HighPressure: 				st_Variable:= IotExtractType(monitor.Cooling.HeatPumpSystem.SecondaryHeatpumpGet.HeatpumpData.r_HighPressure, 1, 0); 
// eDataMappingVarNames.Cooling_HeatPumpSystem_SecondaryHeatpumpGet_HeatpumpData_r_LowPressure: 				st_Variable:= IotExtractType(monitor.Cooling.HeatPumpSystem.SecondaryHeatpumpGet.HeatpumpData.r_LowPressure, 1, 0); 
// eDataMappingVarNames.Cooling_HeatPumpSystem_SecondaryHeatpumpGet_HeatpumpData_r_CompInputTemp: 				st_Variable:= IotExtractType(monitor.Cooling.HeatPumpSystem.SecondaryHeatpumpGet.HeatpumpData.r_CompInputTemp, 1, 0); 
// eDataMappingVarNames.Cooling_HeatPumpSystem_SecondaryHeatpumpGet_HeatpumpData_r_OutdoorTemp: 				st_Variable:= IotExtractType(monitor.Cooling.HeatPumpSystem.SecondaryHeatpumpGet.HeatpumpData.r_OutdoorTemp, 1, 0); 
// eDataMappingVarNames.Cooling_HeatPumpSystem_SecondaryHeatpumpGet_HeatpumpData_r_CompOutputTemp: 				st_Variable:= IotExtractType(monitor.Cooling.HeatPumpSystem.SecondaryHeatpumpGet.HeatpumpData.r_CompOutputTemp, 1, 0); 
// eDataMappingVarNames.Cooling_HeatPumpSystem_SecondaryHeatpumpGet_HeatpumpData_ui_WaterFlowRate: 				st_Variable:= IotExtractType(monitor.Cooling.HeatPumpSystem.SecondaryHeatpumpGet.HeatpumpData.ui_WaterFlowRate, 1, 0); 
// eDataMappingVarNames.Cooling_HeatPumpSystem_SecondaryHeatpumpGet_HeatpumpData_w_ErrorList_1: 				st_Variable:= IotExtractType(monitor.Cooling.HeatPumpSystem.SecondaryHeatpumpGet.HeatpumpData.w_ErrorList[1], 0, 0); 
// eDataMappingVarNames.Cooling_HeatPumpSystem_SecondaryHeatpumpGet_HeatpumpData_w_ErrorList_2: 				st_Variable:= IotExtractType(monitor.Cooling.HeatPumpSystem.SecondaryHeatpumpGet.HeatpumpData.w_ErrorList[2], 0, 0); 
// eDataMappingVarNames.Cooling_HeatPumpSystem_SecondaryHeatpumpGet_HeatpumpData_w_ErrorList_3: 				st_Variable:= IotExtractType(monitor.Cooling.HeatPumpSystem.SecondaryHeatpumpGet.HeatpumpData.w_ErrorList[3], 0, 0); 
// eDataMappingVarNames.Cooling_HeatPumpSystem_SecondaryHeatpumpGet_HeatpumpData_w_ErrorList_4: 				st_Variable:= IotExtractType(monitor.Cooling.HeatPumpSystem.SecondaryHeatpumpGet.HeatpumpData.w_ErrorList[4], 0, 0); 
// eDataMappingVarNames.Cooling_HeatPumpSystem_SecondaryHeatpumpGet_HeatpumpData_w_ErrorList_5: 				st_Variable:= IotExtractType(monitor.Cooling.HeatPumpSystem.SecondaryHeatpumpGet.HeatpumpData.w_ErrorList[5], 0, 0); 
// eDataMappingVarNames.Cooling_HeatPumpSystem_SecondaryHeatpumpGet_HeatpumpData_w_ErrorList_6: 				st_Variable:= IotExtractType(monitor.Cooling.HeatPumpSystem.SecondaryHeatpumpGet.HeatpumpData.w_ErrorList[6], 0, 0); 
// eDataMappingVarNames.Cooling_HeatPumpSystem_SecondaryHeatpumpGet_HeatpumpData_w_ErrorList_7: 				st_Variable:= IotExtractType(monitor.Cooling.HeatPumpSystem.SecondaryHeatpumpGet.HeatpumpData.w_ErrorList[7], 0, 0); 
// eDataMappingVarNames.Cooling_HeatPumpSystem_SecondaryHeatpumpGet_HeatpumpData_r_FanSpeedPCT: 				st_Variable:= IotExtractType(monitor.Cooling.HeatPumpSystem.SecondaryHeatpumpGet.HeatpumpData.r_FanSpeedPCT, 0, 0); 
// eDataMappingVarNames.Cooling_HeatPumpSystem_SecondaryHeatpumpGet_HeatpumpData_r_PumpSpeedPCT: 				st_Variable:= IotExtractType(monitor.Cooling.HeatPumpSystem.SecondaryHeatpumpGet.HeatpumpData.r_PumpSpeedPCT, 0, 0); 
// eDataMappingVarNames.Cooling_HeatPumpSystem_SecondaryHeatpumpGet_HeatpumpData_r_SetpointHeating: 				st_Variable:= IotExtractType(monitor.Cooling.HeatPumpSystem.SecondaryHeatpumpGet.HeatpumpData.r_SetpointHeating, 0, 0); 
// eDataMappingVarNames.Cooling_HeatPumpSystem_SecondaryHeatpumpGet_HeatpumpData_r_SetpointCooling: 				st_Variable:= IotExtractType(monitor.Cooling.HeatPumpSystem.SecondaryHeatpumpGet.HeatpumpData.r_SetpointCooling, 0, 0); 
// eDataMappingVarNames.Cooling_HeatPumpSystem_SecondaryHeatpumpGet_HeatpumpData_b_DefrostingActive: 				st_Variable:= IotExtractType(monitor.Cooling.HeatPumpSystem.SecondaryHeatpumpGet.HeatpumpData.b_DefrostingActive, 0, 0); 
// eDataMappingVarNames.Cooling_Events_b_SystemOvertemperatureWarning: 				st_Variable:= IotExtractType(monitor.Cooling.Events. .b_SystemOvertemperatureWarning, 0, 0); 
// eDataMappingVarNames.Cooling_Events_b_SystemUnderTemperatureWarning: 				st_Variable:= IotExtractType(monitor.Cooling.Events.b_SystemUnderTemperatureWarning, 0, 0); 
// eDataMappingVarNames.Cooling_Events_b_CoolingSystemFuseFailure: 				st_Variable:= IotExtractType(monitor.Cooling.Events.b_CoolingSystemFuseFailure, 0, 0); 
// eDataMappingVarNames.Cooling_Events_b_ACwaterPumpTimeOut: 				st_Variable:= IotExtractType(monitor.Cooling.Events.b_ACwaterPumpTimeOut, 0, 0); 
// eDataMappingVarNames.Cooling_Events_b_InverterLoopValveStuck: 				st_Variable:= IotExtractType(monitor.Cooling.Events.b_InverterLoopValveStuck, 0, 0); 
// eDataMappingVarNames.Cooling_Events_b_BattLoopValveStuck: 				st_Variable:= IotExtractType(monitor.Cooling.Events.b_BattLoopValveStuck, 0, 0); 
// eDataMappingVarNames.Cooling_Events_b_FancoilLoopValveStuck: 				st_Variable:= IotExtractType(monitor.Cooling.Events.b_FancoilLoopValveStuck, 0, 0); 
// eDataMappingVarNames.Cooling_Events_b_DCpumpPressureFault: 				st_Variable:= IotExtractType(monitor.Cooling.Events.b_DCpumpPressureFault, 0, 0); 
// eDataMappingVarNames.Cooling_Events_b_DCpumpTimeout: 				st_Variable:= IotExtractType(monitor.Cooling.Events.b_DCpumpTimeout, 0, 0); 
// eDataMappingVarNames.Cooling_Events_b_CoolingLoopIdlePressureWarning: 				st_Variable:= IotExtractType(monitor.Cooling.Events.b_CoolingLoopIdlePressureWarning, 0, 0); 
// eDataMappingVarNames.Cooling_Events_b_CoolingLoopIdlePressureError: 				st_Variable:= IotExtractType(monitor.Cooling.Events.b_CoolingLoopIdlePressureError, 0, 0); 
// eDataMappingVarNames.Cooling_Events_b_InverterCoolingLoopError: 				st_Variable:= IotExtractType(monitor.Cooling.Events.b_InverterCoolingLoopError, 0, 0); 
// eDataMappingVarNames.Cooling_Events_b_HeatpumpWarning: 				st_Variable:= IotExtractType(monitor.Cooling.Events.b_HeatpumpWarning, 0, 0); 
// eDataMappingVarNames.Cooling_Events_b_HeatPumpError: 				st_Variable:= IotExtractType(monitor.Cooling.Events.b_HeatPumpError, 0, 0); 
// eDataMappingVarNames.Cooling_Events_b_CoolantTempTooLow: 				st_Variable:= IotExtractType(monitor.Cooling.Events.b_CoolantTempTooLow, 0, 0); 
// eDataMappingVarNames.Cooling_Events_b_CoolantTempLow: 				st_Variable:= IotExtractType(monitor.Cooling.Events.b_CoolantTempLow, 0, 0); 
// eDataMappingVarNames.Cooling_Events_b_CoolantTempTooHigh: 				st_Variable:= IotExtractType(monitor.Cooling.Events.b_CoolantTempTooHigh, 0, 0); 
// eDataMappingVarNames.Cooling_Events_b_CoolantTempHigh: 				st_Variable:= IotExtractType(monitor.Cooling.Events.b_CoolantTempHigh, 0, 0); 
// eDataMappingVarNames.Router_Device_SystemUptime: 				st_Variable:= IotExtractType(monitor.Router.Device.SystemUptime, 0, 0); 
// eDataMappingVarNames.Router_Device_Temperature: 				st_Variable:= IotExtractType(monitor.Router.Device.Temperature, 0, 0); 
// eDataMappingVarNames.Router_Device_RouterSerial: 				st_Variable:= IotExtractType(monitor.Router.Device.RouterSerial, 0, 0); 
// eDataMappingVarNames.Router_GPS_Latitude: 				st_Variable:= IotExtractType(monitor.Router.GPS.Latitude, 0, 0); 
// eDataMappingVarNames.Router_GPS_Longitude: 				st_Variable:= IotExtractType(monitor.Router.GPS.Longitude, 0, 0); 
// eDataMappingVarNames.Router_GPS_FixTime: 				st_Variable:= IotExtractType(monitor.Router.GPS.FixTime, 0, 0); 
// eDataMappingVarNames.Router_GPS_DateTime: 				st_Variable:= IotExtractType(monitor.Router.GPS.DateTime, 0, 0); 
// eDataMappingVarNames.Router_GPS_Speed: 				st_Variable:= IotExtractType(monitor.Router.GPS.Speed, 0, 0); 
// eDataMappingVarNames.Router_GPS_SatCount: 				st_Variable:= IotExtractType(monitor.Router.GPS.SatCount, 0, 0); 
// eDataMappingVarNames.Router_GPS_Accuracy: 				st_Variable:= IotExtractType(monitor.Router.GPS.Accuracy, 0, 0); 
// eDataMappingVarNames.Router_Mobile_NetworkOperator: 				st_Variable:= IotExtractType(monitor.Router.Mobile.NetworkOperator, 0, 0); 
// eDataMappingVarNames.Router_Mobile_NetworkInfo: 				st_Variable:= IotExtractType(monitor.Router.Mobile.NetworkInfo, 0, 0); 
// eDataMappingVarNames.Router_Mobile_NetworkType: 				st_Variable:= IotExtractType(monitor.Router.Mobile.NetworkType, 0, 0); 
// eDataMappingVarNames.Router_Mobile_RSSI: 				st_Variable:= IotExtractType(monitor.Router.Mobile.RSSI, 0, 0); 
// eDataMappingVarNames.Router_Mobile_ui_Sim1DataSendMonth: 				st_Variable:= IotExtractType(monitor.Router.Mobile.ui_Sim1DataSendMonth, 0, 0); 
// eDataMappingVarNames.Router_Mobile_ui_Sim1DataReceivedMonth: 				st_Variable:= IotExtractType(monitor.Router.Mobile.ui_Sim1DataReceivedMonth, 0, 0); 
// eDataMappingVarNames.Router_Mobile_ui_Sim2DataSendMonth: 				st_Variable:= IotExtractType(monitor.Router.Mobile.ui_Sim2DataSendMonth, 0, 0); 
// eDataMappingVarNames.Router_Mobile_ui_Sim2DataReceivedMonth: 				st_Variable:= IotExtractType(monitor.Router.Mobile.ui_Sim2DataReceivedMonth, 0, 0); 
// eDataMappingVarNames.Router_Mobile_s_EmergencySMSNumber: 				st_Variable:= IotExtractType(monitor.Router.Mobile.s_EmergencySMSNumber, 0, 0); 
// eDataMappingVarNames.Router_Mobile_s_SecondarySMSNumber: 				st_Variable:= IotExtractType(monitor.Router.Mobile.s_SecondarySMSNumber, 0, 0); 
// eDataMappingVarNames.Router_Mobile_s_EmergencySMSDevName: 				st_Variable:= IotExtractType(monitor.Router.Mobile.s_EmergencySMSDevName, 0, 0); 
// eDataMappingVarNames.Router_Mobile_st_LatestSMSMessage: 				st_Variable:= IotExtractType(monitor.Router.Mobile.st_LatestSMSMessage, 0, 0); 
// eDataMappingVarNames.Router_Mobile_ModemState: 				st_Variable:= IotExtractType(monitor.Router.Mobile.ModemState, 0, 0); 
// eDataMappingVarNames.Router_Mobile_NetworkState: 				st_Variable:= IotExtractType(monitor.Router.Mobile.NetworkState, 0, 0); 
// eDataMappingVarNames.Router_Mobile_ui_ActiveSim: 				st_Variable:= IotExtractType(monitor.Router.Mobile.ui_ActiveSim, 0, 0); 
// eDataMappingVarNames.Router_Mobile_SimStatus: 				st_Variable:= IotExtractType(monitor.Router.Mobile.SimStatus, 0, 0); 
// eDataMappingVarNames.Router_Wifi_WifiClienModeStatus: 				st_Variable:= IotExtractType(monitor.Router.Wifi.WifiClienModeStatus, 0, 0); 
// eDataMappingVarNames.Router_Wifi_WifiAPModeStatus: 				st_Variable:= IotExtractType(monitor.Router.Wifi.WifiAPModeStatus, 0, 0); 
// eDataMappingVarNames.Router_Wifi_WifiApNumberOfClients: 				st_Variable:= IotExtractType(monitor.Router.Wifi.WifiApNumberOfClients, 0, 0); 
// eDataMappingVarNames.Router_e_SMSStatus: 				st_Variable:= IotExtractType(monitor.Router.e_SMSStatus, 0, 0); 
// eDataMappingVarNames.Router_Events_b_MBCommWarning: 				st_Variable:= IotExtractType(monitor.Router.Events.b_MBCommWarning, 0, 0); 
// eDataMappingVarNames.Router_Events_b_NoSimWarning: 				st_Variable:= IotExtractType(monitor.Router.Events.b_NoSimWarning, 0, 0); 
// eDataMappingVarNames.Router_Events_b_NoNetworkWarning: 				st_Variable:= IotExtractType(monitor.Router.Events.b_NoNetworkWarning, 0, 0); 
// eDataMappingVarNames.Router_Events_b_noGPSFixWarning: 				st_Variable:= IotExtractType(monitor.Router.Events.b_noGPSFixWarning, 0, 0); 
// eDataMappingVarNames.Router_Events_b_SMSNotSendError: 				st_Variable:= IotExtractType(monitor.Router.Events.b_SMSNotSendError, 0, 0); 
// eDataMappingVarNames.Router_Events_b_NoSMSNumberAvailable: 				st_Variable:= IotExtractType(monitor.Router.Events.b_NoSMSNumberAvailable, 0, 0); 
// eDataMappingVarNames.Router_Events_b_TimeUpdateFailed: 				st_Variable:= IotExtractType(monitor.Router.Events.b_TimeUpdateFailed, 0, 0); 
// eDataMappingVarNames.controlfb_control_b_start: 															st_Variable:= IotExtractType(controlvars.control.b_start, 0, 0); 
// eDataMappingVarNames.controlfb_control_b_stop: 																st_Variable:= IotExtractType(controlvars.control.b_stop, 0, 0); 
// eDataMappingVarNames.controlfb_control_b_shutdown: 															st_Variable:= IotExtractType(controlvars.control.b_shutdown, 0, 0); 
// eDataMappingVarNames.controlfb_control_b_Reset: 															st_Variable:= IotExtractType(controlvars.control.b_Reset, 0, 0); 
// eDataMappingVarNames.controlfb_control_b_SystemShutdown: 													st_Variable:= IotExtractType(controlvars.control.b_SystemShutdown, 0, 0); 
// eDataMappingVarNames.controlfb_control_b_EMstop: 															st_Variable:= IotExtractType(controlvars.control.b_EMstop, 0, 0); 
// eDataMappingVarNames.controlfb_control_b_ClearHistory: 														st_Variable:= IotExtractType(controlvars.control.b_ClearHistory, 0, 0); 
// eDataMappingVarNames.controlfb_control_b_ActivateSettings: 													st_Variable:= IotExtractType(controlvars.control.b_ActivateSettings, 0, 0); 
// eDataMappingVarNames.controlfb_control_b_startDeHum: 														st_Variable:= IotExtractType(controlvars.control.b_startDeHum, 0, 0); 
// eDataMappingVarNames.controlfb_Operation_inputgrid_b_SyncClose: 											st_Variable:= IotExtractType(controlvars.Operation.inputgrid.b_SyncClose, 0, 0); 
// eDataMappingVarNames.controlfb_Operation_Genset_b_manualStart: 												st_Variable:= IotExtractType(controlvars.Operation.Genset.b_manualStart, 0, 0); 
// eDataMappingVarNames.controlfb_Operation_PSB_b_SyncClose: 													st_Variable:= IotExtractType(controlvars.Operation.PSB.b_SyncClose, 0, 0); 
// eDataMappingVarNames.controlfb_Operation_charger_b_StartCharging: 											st_Variable:= IotExtractType(controlvars.Operation.charger.b_StartCharging, 0, 0); 
// eDataMappingVarNames.controlfb_Operation_charger_b_ResetCharger: 											st_Variable:= IotExtractType(controlvars.Operation.charger.b_ResetCharger, 0, 0); 
// eDataMappingVarNames.controlfb_Operation_system_r_NominalVoltage: 											st_Variable:= IotExtractType(controlvars.Operation.system.r_NominalVoltage, 0, 0); 
// eDataMappingVarNames.controlfb_Operation_system_r_NominalFrequency: 										st_Variable:= IotExtractType(controlvars.Operation.system.r_NominalFrequency, 0, 0); 
// eDataMappingVarNames.controlfb_Operation_system_r_Pset: 													st_Variable:= IotExtractType(controlvars.Operation.system.r_Pset, 0, 0); 
// eDataMappingVarNames.controlfb_Operation_system_r_Qset: 													st_Variable:= IotExtractType(controlvars.Operation.system.r_Qset, 0, 0); 
// eDataMappingVarNames.controlfb_Operation_system_r_PFset: 													st_Variable:= IotExtractType(controlvars.Operation.system.r_PFset, 0, 0); 
// eDataMappingVarNames.controlfb_Operation_system_b_PFsetEnable: 												st_Variable:= IotExtractType(controlvars.Operation.system.b_PFsetEnable, 0, 0); 
// eDataMappingVarNames.controlfb_Operation_system_b_SounderMute: 												st_Variable:= IotExtractType(controlvars.Operation.system.b_SounderMute, 0, 0); 
// eDataMappingVarNames.controlfb_Operation_system_b_SounderTest: 												st_Variable:= IotExtractType(controlvars.Operation.system.b_SounderTest, 0, 0); 
// eDataMappingVarNames.controlfb_Operation_system_b_GenGridModeTrans: 										st_Variable:= IotExtractType(controlvars.Operation.system.b_GenGridModeTrans, 0, 0); 
// eDataMappingVarNames.controlfb_Operation_system_b_GridTakeOverEnable: 										st_Variable:= IotExtractType(controlvars.Operation.system.b_GridTakeOverEnable, 0, 0); 
// eDataMappingVarNames.controlfb_Operation_parallel_b_DetectSlaves: 											st_Variable:= IotExtractType(controlvars.Operation.parallel.b_DetectSlaves, 0, 0); 
// eDataMappingVarNames.controlfb_Operation_parallel_r_ActivePowerSlave1: 										st_Variable:= IotExtractType(controlvars.Operation.parallel.r_ActivePowerSlave1, 0, 0); 
// eDataMappingVarNames.controlfb_Operation_parallel_r_ReactivePowerSlave1: 									st_Variable:= IotExtractType(controlvars.Operation.parallel.r_ReactivePowerSlave1, 0, 0); 
// eDataMappingVarNames.controlfb_Operation_parallel_r_ActivePowerSlave2: 										st_Variable:= IotExtractType(controlvars.Operation.parallel.r_ActivePowerSlave2, 0, 0); 
// eDataMappingVarNames.controlfb_Operation_parallel_r_ReactivePowerSlave2: 									st_Variable:= IotExtractType(controlvars.Operation.parallel.r_ReactivePowerSlave2, 0, 0); 
// eDataMappingVarNames.controlfb_Operation_BMS_b_ManualStartHVDC: 											st_Variable:= IotExtractType(controlvars.Operation.BMS.b_ManualStartHVDC, 0, 0); 
// eDataMappingVarNames.controlfb_SoftSettings_inputgrid_PeakshaveMode: 										st_Variable:= IotExtractType(controlvars.SoftSettings.inputgrid.PeakshaveMode, 0, 0); 
// eDataMappingVarNames.controlfb_SoftSettings_inputgrid_setpointTimeslot1_r_SocTarget:		 				st_Variable:= IotExtractType(controlvars.SoftSettings.inputgrid.setpointTimeslot1.r_SocTarget, 0, 0); 
// eDataMappingVarNames.controlfb_SoftSettings_inputgrid_setpointTimeslot1_r_IdleChargePower: 					st_Variable:= IotExtractType(controlvars.SoftSettings.inputgrid.setpointTimeslot1.r_IdleChargePower, 0, 0); 
// eDataMappingVarNames.controlfb_SoftSettings_inputgrid_setpointTimeslot1_r_FeedInCurrentLimitSoft: 			st_Variable:= IotExtractType(controlvars.SoftSettings.inputgrid.setpointTimeslot1.r_FeedInCurrentLimitSoft, 0, 0); 
// eDataMappingVarNames.controlfb_SoftSettings_inputgrid_setpointTimeslot1_r_SupplyCurrentLimitSoft: 			st_Variable:= IotExtractType(controlvars.SoftSettings.inputgrid.setpointTimeslot1.r_SupplyCurrentLimitSoft, 0, 0); 
// eDataMappingVarNames.controlfb_SoftSettings_inputgrid_setpointTimeslot2_r_SocTarget: 						st_Variable:= IotExtractType(controlvars.SoftSettings.inputgrid.setpointTimeslot2.r_SocTarget, 0, 0); 
// eDataMappingVarNames.controlfb_SoftSettings_inputgrid_setpointTimeslot2_r_IdleChargePower: 					st_Variable:= IotExtractType(controlvars.SoftSettings.inputgrid.setpointTimeslot2.r_IdleChargePower, 0, 0); 
// eDataMappingVarNames.controlfb_SoftSettings_inputgrid_setpointTimeslot2_r_FeedInCurrentLimitSoft: 			st_Variable:= IotExtractType(controlvars.SoftSettings.inputgrid.setpointTimeslot2.r_FeedInCurrentLimitSoft, 0, 0); 
// eDataMappingVarNames.controlfb_SoftSettings_inputgrid_setpointTimeslot2_r_SupplyCurrentLimitSoft: 			st_Variable:= IotExtractType(controlvars.SoftSettings.inputgrid.setpointTimeslot2.r_SupplyCurrentLimitSoft, 0, 0); 
// eDataMappingVarNames.controlfb_SoftSettings_inputgrid_b_BreakerControl: 									st_Variable:= IotExtractType(controlvars.SoftSettings.inputgrid.b_BreakerControl, 0, 0); 
// eDataMappingVarNames.controlfb_SoftSettings_inputgrid_b_ReverseCTDirection: 								st_Variable:= IotExtractType(controlvars.SoftSettings.inputgrid.b_ReverseCTDirection, 0, 0); 
// eDataMappingVarNames.controlfb_SoftSettings_inputgrid_ui_CTrange: 											st_Variable:= IotExtractType(controlvars.SoftSettings.inputgrid.ui_CTrange, 0, 0); 
// eDataMappingVarNames.controlfb_SoftSettings_inputgrid_r_VTratio: 											st_Variable:= IotExtractType(controlvars.SoftSettings.inputgrid.r_VTratio, 0, 0); 
// eDataMappingVarNames.controlfb_SoftSettings_inputgrid_b_GridCodesActive: 									st_Variable:= IotExtractType(controlvars.SoftSettings.inputgrid.b_GridCodesActive, 0, 0); 
// eDataMappingVarNames.controlfb_SoftSettings_inputgrid_b_WeakGridInput: 										st_Variable:= IotExtractType(controlvars.SoftSettings.inputgrid.b_WeakGridInput, 0, 0); 
// eDataMappingVarNames.controlfb_SoftSettings_inputgrid_breaker_AutoConnect: 									st_Variable:= IotExtractType(controlvars.SoftSettings.inputgrid.breaker.AutoConnect, 0, 0); 
// eDataMappingVarNames.controlfb_SoftSettings_inputgrid_breaker_ShutdownDisconnect: 							st_Variable:= IotExtractType(controlvars.SoftSettings.inputgrid.breaker.ShutdownDisconnect, 0, 0); 
// eDataMappingVarNames.controlfb_SoftSettings_inputgrid_breaker_EMstopDisconnect: 							st_Variable:= IotExtractType(controlvars.SoftSettings.inputgrid.breaker.EMstopDisconnect, 0, 0); 
// eDataMappingVarNames.controlfb_SoftSettings_inputgrid_breaker_CurrentLimitDisconnect: 						st_Variable:= IotExtractType(controlvars.SoftSettings.inputgrid.breaker.CurrentLimitDisconnect, 0, 0); 
// eDataMappingVarNames.controlfb_SoftSettings_inputgrid_breaker_CurrentLimitRetries: 							st_Variable:= IotExtractType(controlvars.SoftSettings.inputgrid.breaker.CurrentLimitRetries, 0, 0); 
// eDataMappingVarNames.controlfb_SoftSettings_inputgenset_b_AutoStartStop: 									st_Variable:= IotExtractType(controlvars.SoftSettings.inputgenset.b_AutoStartStop, 0, 0); 
// eDataMappingVarNames.controlfb_SoftSettings_inputgenset_b_HydridMode: 										st_Variable:= IotExtractType(controlvars.SoftSettings.inputgenset.b_HydridMode, 0, 0); 
// eDataMappingVarNames.controlfb_SoftSettings_inputgenset_b_EnableSchedule: 									st_Variable:= IotExtractType(controlvars.SoftSettings.inputgenset.b_EnableSchedule, 0, 0); 
// eDataMappingVarNames.controlfb_SoftSettings_inputgenset_setpointTimeslot1_r_SoCStart: 						st_Variable:= IotExtractType(controlvars.SoftSettings.inputgenset.setpointTimeslot1.r_SoCStart, 0, 0); 
// eDataMappingVarNames.controlfb_SoftSettings_inputgenset_setpointTimeslot1_r_SoCStop: 						st_Variable:= IotExtractType(controlvars.SoftSettings.inputgenset.setpointTimeslot1.r_SoCStop, 0, 0); 
// eDataMappingVarNames.controlfb_SoftSettings_inputgenset_setpointTimeslot1_r_BatteryloadStart: 				st_Variable:= IotExtractType(controlvars.SoftSettings.inputgenset.setpointTimeslot1.r_BatteryloadStart, 0, 0); 
// eDataMappingVarNames.controlfb_SoftSettings_inputgenset_setpointTimeslot1_r_BatteryloadStop: 				st_Variable:= IotExtractType(controlvars.SoftSettings.inputgenset.setpointTimeslot1.r_BatteryloadStop, 0, 0); 
// eDataMappingVarNames.controlfb_SoftSettings_inputgenset_setpointTimeslot1_b_StartAtBatteryError: 			st_Variable:= IotExtractType(controlvars.SoftSettings.inputgenset.setpointTimeslot1.b_StartAtBatteryError, 0, 0); 
// eDataMappingVarNames.controlfb_SoftSettings_inputgenset_setpointTimeslot2_r_SoCStart: 						st_Variable:= IotExtractType(controlvars.SoftSettings.inputgenset.setpointTimeslot2.r_SoCStart, 0, 0); 
// eDataMappingVarNames.controlfb_SoftSettings_inputgenset_setpointTimeslot2_r_SoCStop: 						st_Variable:= IotExtractType(controlvars.SoftSettings.inputgenset.setpointTimeslot2.r_SoCStop, 0, 0); 
// eDataMappingVarNames.controlfb_SoftSettings_inputgenset_setpointTimeslot2_r_BatteryloadStart: 				st_Variable:= IotExtractType(controlvars.SoftSettings.inputgenset.setpointTimeslot2.r_BatteryloadStart, 0, 0); 
// eDataMappingVarNames.controlfb_SoftSettings_inputgenset_setpointTimeslot2_r_BatteryloadStop: 				st_Variable:= IotExtractType(controlvars.SoftSettings.inputgenset.setpointTimeslot2.r_BatteryloadStop, 0, 0); 
// eDataMappingVarNames.controlfb_SoftSettings_inputgenset_setpointTimeslot2_b_StartAtBatteryError: 			st_Variable:= IotExtractType(controlvars.SoftSettings.inputgenset.setpointTimeslot2.b_StartAtBatteryError, 0, 0); 
// eDataMappingVarNames.controlfb_SoftSettings_inputgenset_b_PSBExtGensetMonitoring: 							st_Variable:= IotExtractType(controlvars.SoftSettings.inputgenset.b_PSBExtGensetMonitoring, 0, 0); 
// eDataMappingVarNames.controlfb_SoftSettings_inputgenset_b_FreqProtectionEnable: 							st_Variable:= IotExtractType(controlvars.SoftSettings.inputgenset.b_FreqProtectionEnable, 0, 0); 
// eDataMappingVarNames.controlfb_SoftSettings_inputgenset_Generator_e_GensetMode: 							st_Variable:= IotExtractType(controlvars.SoftSettings.inputgenset.Generator.e_GensetMode, 0, 0); 
// eDataMappingVarNames.controlfb_SoftSettings_inputgenset_Generator_b_GensetLoadshareLine: 					st_Variable:= IotExtractType(controlvars.SoftSettings.inputgenset.Generator.b_GensetLoadshareLine, 0, 0); 
// eDataMappingVarNames.controlfb_SoftSettings_inputgenset_Generator_r_RatedPower: 							st_Variable:= IotExtractType(controlvars.SoftSettings.inputgenset.Generator.r_RatedPower, 0, 0); 
// eDataMappingVarNames.controlfb_SoftSettings_inputgenset_Generator_r_powerloadMax: 							st_Variable:= IotExtractType(controlvars.SoftSettings.inputgenset.Generator.r_powerloadMax, 0, 0); 
// eDataMappingVarNames.controlfb_SoftSettings_inputgenset_Generator_r_PowerloadMin: 							st_Variable:= IotExtractType(controlvars.SoftSettings.inputgenset.Generator.r_PowerloadMin, 0, 0); 
// eDataMappingVarNames.controlfb_SoftSettings_inputgenset_Generator_r_PowerloadEff: 							st_Variable:= IotExtractType(controlvars.SoftSettings.inputgenset.Generator.r_PowerloadEff, 0, 0); 
// eDataMappingVarNames.controlfb_SoftSettings_inputgenset_Generator_r_ramprate: 								st_Variable:= IotExtractType(controlvars.SoftSettings.inputgenset.Generator.r_ramprate, 0, 0); 
// eDataMappingVarNames.controlfb_SoftSettings_inputgenset_Generator_ui_CooldownTime: 							st_Variable:= IotExtractType(controlvars.SoftSettings.inputgenset.Generator.ui_CooldownTime, 0, 0); 
// eDataMappingVarNames.controlfb_SoftSettings_inputgenset_Generator_ui_WarmupTime: 							st_Variable:= IotExtractType(controlvars.SoftSettings.inputgenset.Generator.ui_WarmupTime, 0, 0); 
// eDataMappingVarNames.controlfb_SoftSettings_inputgenset_Loadbank_b_Enable: 									st_Variable:= IotExtractType(controlvars.SoftSettings.inputgenset.Loadbank.b_Enable, 0, 0); 
// eDataMappingVarNames.controlfb_SoftSettings_inputgenset_Loadbank_r_PowerRating: 							st_Variable:= IotExtractType(controlvars.SoftSettings.inputgenset.Loadbank.r_PowerRating, 0, 0); 
// eDataMappingVarNames.controlfb_SoftSettings_inputgenset_Loadbank_r_PowerStepSize: 							st_Variable:= IotExtractType(controlvars.SoftSettings.inputgenset.Loadbank.r_PowerStepSize, 0, 0); 
// eDataMappingVarNames.controlfb_SoftSettings_PSB_PeakshaveMode: 												st_Variable:= IotExtractType(controlvars.SoftSettings.PSB.PeakshaveMode, 0, 0); 
// eDataMappingVarNames.controlfb_SoftSettings_PSB_setpointTimeslot1_r_SocTarget: 								st_Variable:= IotExtractType(controlvars.SoftSettings.PSB.setpointTimeslot1.r_SocTarget, 0, 0); 
// eDataMappingVarNames.controlfb_SoftSettings_PSB_setpointTimeslot1_r_IdleChargePower: 						st_Variable:= IotExtractType(controlvars.SoftSettings.PSB.setpointTimeslot1.r_IdleChargePower, 0, 0); 
// eDataMappingVarNames.controlfb_SoftSettings_PSB_setpointTimeslot1_r_FeedInCurrentLimitSoft: 				st_Variable:= IotExtractType(controlvars.SoftSettings.PSB.setpointTimeslot1.r_FeedInCurrentLimitSoft, 0, 0); 
// eDataMappingVarNames.controlfb_SoftSettings_PSB_setpointTimeslot1_r_SupplyCurrentLimitSoft: 				st_Variable:= IotExtractType(controlvars.SoftSettings.PSB.setpointTimeslot1.r_SupplyCurrentLimitSoft, 0, 0); 
// eDataMappingVarNames.controlfb_SoftSettings_PSB_setpointTimeslot2_r_SocTarget: 								st_Variable:= IotExtractType(controlvars.SoftSettings.PSB.setpointTimeslot2.r_SocTarget, 0, 0); 
// eDataMappingVarNames.controlfb_SoftSettings_PSB_setpointTimeslot2_r_IdleChargePower: 						st_Variable:= IotExtractType(controlvars.SoftSettings.PSB.setpointTimeslot2.r_IdleChargePower, 0, 0); 
// eDataMappingVarNames.controlfb_SoftSettings_PSB_setpointTimeslot2_r_FeedInCurrentLimitSoft: 				st_Variable:= IotExtractType(controlvars.SoftSettings.PSB.setpointTimeslot2.r_FeedInCurrentLimitSoft, 0, 0); 
// eDataMappingVarNames.controlfb_SoftSettings_PSB_setpointTimeslot2_r_SupplyCurrentLimitSoft: 				st_Variable:= IotExtractType(controlvars.SoftSettings.PSB.setpointTimeslot2.r_SupplyCurrentLimitSoft, 0, 0); 
// eDataMappingVarNames.controlfb_SoftSettings_PSB_b_BreakerControl: 											st_Variable:= IotExtractType(controlvars.SoftSettings.PSB.b_BreakerControl, 0, 0); 
// eDataMappingVarNames.controlfb_SoftSettings_PSB_b_ReverseCTDirection: 										st_Variable:= IotExtractType(controlvars.SoftSettings.PSB.b_ReverseCTDirection, 0, 0); 
// eDataMappingVarNames.controlfb_SoftSettings_PSB_ui_CTrange: 												st_Variable:= IotExtractType(controlvars.SoftSettings.PSB.ui_CTrange, 0, 0); 
// eDataMappingVarNames.controlfb_SoftSettings_PSB_r_VTratio: 													st_Variable:= IotExtractType(controlvars.SoftSettings.PSB.r_VTratio, 0, 0); 
// eDataMappingVarNames.controlfb_SoftSettings_system_b_EnableSchedule: 										st_Variable:= IotExtractType(controlvars.SoftSettings.system.b_EnableSchedule, 0, 0); 
// eDataMappingVarNames.controlfb_SoftSettings_system_b_EnableTransportMode: 									st_Variable:= IotExtractType(controlvars.SoftSettings.system.b_EnableTransportMode, 0, 0); 
// eDataMappingVarNames.controlfb_SoftSettings_system_b_EcoModeEnable: 										st_Variable:= IotExtractType(controlvars.SoftSettings.system.b_EcoModeEnable, 0, 0); 
// eDataMappingVarNames.controlfb_SoftSettings_system_e_UgridPowerMode: 										st_Variable:= IotExtractType(controlvars.SoftSettings.system.e_UgridPowerMode, 0, 0); 
// eDataMappingVarNames.controlfb_SoftSettings_system_e_NetcontactorMode: 										st_Variable:= IotExtractType(controlvars.SoftSettings.system.e_NetcontactorMode, 0, 0); 
// eDataMappingVarNames.controlfb_SoftSettings_system_e_UgridPowerLimitingMode: 								st_Variable:= IotExtractType(controlvars.SoftSettings.system.e_UgridPowerLimitingMode, 0, 0); 
// eDataMappingVarNames.controlfb_SoftSettings_system_b_AutomaticSwitching: 									st_Variable:= IotExtractType(controlvars.SoftSettings.system.b_AutomaticSwitching, 0, 0); 
// eDataMappingVarNames.controlfb_SoftSettings_system_b_AMF: 													st_Variable:= IotExtractType(controlvars.SoftSettings.system.b_AMF, 0, 0); 
// eDataMappingVarNames.controlfb_SoftSettings_system_r_FrequencyDroop: 										st_Variable:= IotExtractType(controlvars.SoftSettings.system.r_FrequencyDroop, 0, 0); 
// eDataMappingVarNames.controlfb_SoftSettings_system_r_VoltageDroop: 											st_Variable:= IotExtractType(controlvars.SoftSettings.system.r_VoltageDroop, 0, 0); 
// eDataMappingVarNames.controlfb_SoftSettings_system_r_SocMin: 												st_Variable:= IotExtractType(controlvars.SoftSettings.system.r_SocMin, 0, 0); 
// eDataMappingVarNames.controlfb_SoftSettings_system_r_SocMax: 												st_Variable:= IotExtractType(controlvars.SoftSettings.system.r_SocMax, 0, 0); 
// eDataMappingVarNames.controlfb_SoftSettings_system_r_PDischargeLimit: 										st_Variable:= IotExtractType(controlvars.SoftSettings.system.r_PDischargeLimit, 0, 0); 
// eDataMappingVarNames.controlfb_SoftSettings_system_r_PChargeLimit: 											st_Variable:= IotExtractType(controlvars.SoftSettings.system.r_PChargeLimit, 0, 0); 
// eDataMappingVarNames.controlfb_SoftSettings_system_r_AMax: 													st_Variable:= IotExtractType(controlvars.SoftSettings.system.r_AMax, 0, 0); 
// eDataMappingVarNames.controlfb_SoftSettings_system_s_SystemName: 											st_Variable:= IotExtractType(controlvars.SoftSettings.system.s_SystemName, 0, 0); 
// eDataMappingVarNames.controlfb_SoftSettings_system_s_SMSnumber: 											st_Variable:= IotExtractType(controlvars.SoftSettings.system.s_SMSnumber, 0, 0); 
// eDataMappingVarNames.controlfb_SoftSettings_system_ScheduleTimeSlot1_b_active: 								st_Variable:= IotExtractType(controlvars.SoftSettings.system.ScheduleTimeSlot1.b_active, 0, 0); 
// eDataMappingVarNames.controlfb_SoftSettings_system_ScheduleTimeSlot1_usi_DayOfWeek: 						st_Variable:= IotExtractType(controlvars.SoftSettings.system.ScheduleTimeSlot1.usi_DayOfWeek, 0, 0); 
// eDataMappingVarNames.controlfb_SoftSettings_system_ScheduleTimeSlot1_usi_HourOfDay: 						st_Variable:= IotExtractType(controlvars.SoftSettings.system.ScheduleTimeSlot1.usi_HourOfDay, 0, 0); 
// eDataMappingVarNames.controlfb_SoftSettings_system_ScheduleTimeSlot1_usi_MinuteOfHour: 						st_Variable:= IotExtractType(controlvars.SoftSettings.system.ScheduleTimeSlot1.usi_MinuteOfHour, 0, 0); 
// eDataMappingVarNames.controlfb_SoftSettings_system_ScheduleTimeSlot2_b_active: 								st_Variable:= IotExtractType(controlvars.SoftSettings.system.ScheduleTimeSlot2.b_active, 0, 0); 
// eDataMappingVarNames.controlfb_SoftSettings_system_ScheduleTimeSlot2_usi_DayOfWeek: 						st_Variable:= IotExtractType(controlvars.SoftSettings.system.ScheduleTimeSlot2.usi_DayOfWeek, 0, 0); 
// eDataMappingVarNames.controlfb_SoftSettings_system_ScheduleTimeSlot2_usi_HourOfDay: 						st_Variable:= IotExtractType(controlvars.SoftSettings.system.ScheduleTimeSlot2.usi_HourOfDay, 0, 0); 
// eDataMappingVarNames.controlfb_SoftSettings_system_ScheduleTimeSlot2_usi_MinuteOfHour: 						st_Variable:= IotExtractType(controlvars.SoftSettings.system.ScheduleTimeSlot2.usi_MinuteOfHour, 0, 0); 
// eDataMappingVarNames.controlfb_SoftSettings_system_by_LEDbrightness: 										st_Variable:= IotExtractType(controlvars.SoftSettings.system.by_LEDbrightness, 0, 0); 
// eDataMappingVarNames.controlfb_SoftSettings_setup_e_AcInputType: 											st_Variable:= IotExtractType(controlvars.SoftSettings.setup.e_AcInputType, 0, 0); 
// eDataMappingVarNames.controlfb_SoftSettings_setup_b_MasterSlaveMode: 										st_Variable:= IotExtractType(controlvars.SoftSettings.setup.b_MasterSlaveMode, 0, 0); 
// eDataMappingVarNames.controlfb_SoftSettings_setup_b_PeakshaveBoxEnable: 									st_Variable:= IotExtractType(controlvars.SoftSettings.setup.b_PeakshaveBoxEnable, 0, 0); 
// eDataMappingVarNames.controlfb_SoftSettings_setup_e_Gridmode: 												st_Variable:= IotExtractType(controlvars.SoftSettings.setup.e_Gridmode, 0, 0); 
// eDataMappingVarNames.controlfb_SoftSettings_setup_e_DcCouplingType: 										st_Variable:= IotExtractType(controlvars.SoftSettings.setup.e_DcCouplingType, 0, 0); 
// eDataMappingVarNames.controlfb_SoftSettings_setup_b_ExtGenset: 												st_Variable:= IotExtractType(controlvars.SoftSettings.setup.b_ExtGenset, 0, 0); 
// eDataMappingVarNames.controlfb_HardSettings_setup_e_ControlSource: 											st_Variable:= IotExtractType(controlvars.HardSettings.setup.e_ControlSource, 0, 0); 
// eDataMappingVarNames.controlfb_HardSettings_charger_r_PowerMax: 											st_Variable:= IotExtractType(controlvars.HardSettings.charger.r_PowerMax, 0, 0); 
// eDataMappingVarNames.controlfb_HardSettings_parallel_b_MasterSlaveEnabled: 									st_Variable:= IotExtractType(controlvars.HardSettings.parallel.b_MasterSlaveEnabled, 0, 0); 
// eDataMappingVarNames.controlfb_HardSettings_parallel_b_UnitIsMaster: 										st_Variable:= IotExtractType(controlvars.HardSettings.parallel.b_UnitIsMaster, 0, 0); 
// eDataMappingVarNames.controlfb_HardSettings_parallel_b_ShutdownOnCommError: 								st_Variable:= IotExtractType(controlvars.HardSettings.parallel.b_ShutdownOnCommError, 0, 0); 
// eDataMappingVarNames.controlfb_HardSettings_parallel_b_EffiencyMode: 										st_Variable:= IotExtractType(controlvars.HardSettings.parallel.b_EffiencyMode, 0, 0); 
// eDataMappingVarNames.controlfb_HardSettings_parallel_r_VoltageDroop: 										st_Variable:= IotExtractType(controlvars.HardSettings.parallel.r_VoltageDroop, 0, 0); 
// eDataMappingVarNames.controlfb_HardSettings_parallel_r_FrequencyDroop: 										st_Variable:= IotExtractType(controlvars.HardSettings.parallel.r_FrequencyDroop, 0, 0); 
// eDataMappingVarNames.controlfb_HardSettings_system_r_PDischargeLimit: 										st_Variable:= IotExtractType(controlvars.HardSettings.system.r_PDischargeLimit, 0, 0); 
// eDataMappingVarNames.controlfb_HardSettings_system_r_PChargeLimit: 											st_Variable:= IotExtractType(controlvars.HardSettings.system.r_PChargeLimit, 0, 0); 
// eDataMappingVarNames.controlfb_HardSettings_system_r_SMax: 													st_Variable:= IotExtractType(controlvars.HardSettings.system.r_SMax, 0, 0); 
// eDataMappingVarNames.controlfb_HardSettings_system_r_Amax: 													st_Variable:= IotExtractType(controlvars.HardSettings.system.r_Amax, 0, 0); 
// eDataMappingVarNames.controlfb_HardSettings_system_e_EarthingSystem: 										st_Variable:= IotExtractType(controlvars.HardSettings.system.e_EarthingSystem, 0, 0); 
// eDataMappingVarNames.controlfb_HardSettings_system_a_ui_InputCurrentLimit_1: 								st_Variable:= IotExtractType(controlvars.HardSettings.system.a_ui_InputCurrentLimit[1], 0, 0); 
// eDataMappingVarNames.controlfb_HardSettings_system_a_ui_InputCurrentLimit_2: 								st_Variable:= IotExtractType(controlvars.HardSettings.system.a_ui_InputCurrentLimit[2], 0, 0); 
// eDataMappingVarNames.controlfb_HardSettings_system_a_ui_OutputCurrentLimit_1: 								st_Variable:= IotExtractType(controlvars.HardSettings.system.a_ui_OutputCurrentLimit[1], 0, 0); 
// eDataMappingVarNames.controlfb_HardSettings_system_a_ui_OutputCurrentLimit_2: 								st_Variable:= IotExtractType(controlvars.HardSettings.system.a_ui_OutputCurrentLimit[2], 0, 0); 
// eDataMappingVarNames.controlfb_HardSettings_system_a_ui_OutputCurrentLimit_3: 								st_Variable:= IotExtractType(controlvars.HardSettings.system.a_ui_OutputCurrentLimit[3], 0, 0); 
// eDataMappingVarNames.Generator_CommunicationOK: 				st_Variable:= IotExtractType(monitor.Generator.CommunicationOK, 0, 0); 
// eDataMappingVarNames.Generator_FuelLow: 				st_Variable:= IotExtractType(monitor.Generator.FuelLow, 0, 0); 
// eDataMappingVarNames.Generator_FuelCritical: 				st_Variable:= IotExtractType(monitor.Generator.FuelCritical, 0, 0); 
// eDataMappingVarNames.Generator_bGenBreakerClosed: 				st_Variable:= IotExtractType(monitor.Generator.bGenBreakerClosed, 0, 0); 
// eDataMappingVarNames.Generator_bMainBreakerClosed: 				st_Variable:= IotExtractType(monitor.Generator.bMainBreakerClosed, 0, 0); 
// eDataMappingVarNames.Generator_bGenRunning: 				st_Variable:= IotExtractType(monitor.Generator.bGenRunning, 0, 0); 
// eDataMappingVarNames.Generator_bGenVoltFreqOK: 				st_Variable:= IotExtractType(monitor.Generator.bGenVoltFreqOK, 0, 0); 
// eDataMappingVarNames.Generator_bMainsFailure: 				st_Variable:= IotExtractType(monitor.Generator.bMainsFailure, 0, 0); 
// eDataMappingVarNames.Generator_eActiveGenMode: 				st_Variable:= IotExtractType(monitor.Generator.eActiveGenMode, 0, 0); 
// eDataMappingVarNames.Generator_bIslandModeActive: 				st_Variable:= IotExtractType(monitor.Generator.bIslandModeActive, 0, 0); 
// eDataMappingVarNames.Generator_bAMFActive: 				st_Variable:= IotExtractType(monitor.Generator.bAMFActive, 0, 0); 
// eDataMappingVarNames.Generator_bPeakshaveActive: 				st_Variable:= IotExtractType(monitor.Generator.bPeakshaveActive, 0, 0); 
// eDataMappingVarNames.Generator_bFixedPowerActive: 				st_Variable:= IotExtractType(monitor.Generator.bFixedPowerActive, 0, 0); 
// eDataMappingVarNames.Generator_ar_LineVoltage_AVG: 				st_Variable:= IotExtractType(monitor.Generator.ar_LineVoltage[0], 1, 1); 
// eDataMappingVarNames.Generator_ar_LineVoltage_L1: 				st_Variable:= IotExtractType(monitor.Generator.ar_LineVoltage[1], 1, 1); 
// eDataMappingVarNames.Generator_ar_LineVoltage_L2: 				st_Variable:= IotExtractType(monitor.Generator.ar_LineVoltage[2], 1, 1); 
// eDataMappingVarNames.Generator_ar_LineVoltage_L3: 				st_Variable:= IotExtractType(monitor.Generator.ar_LineVoltage[3], 1, 1); 
// eDataMappingVarNames.Generator_ar_PhaseVoltage_AVG: 				st_Variable:= IotExtractType(monitor.Generator.ar_PhaseVoltage[0], 1, 1); 
// eDataMappingVarNames.Generator_ar_PhaseVoltage_L1: 				st_Variable:= IotExtractType(monitor.Generator.ar_PhaseVoltage[1], 1, 1); 
// eDataMappingVarNames.Generator_ar_PhaseVoltage_L2: 				st_Variable:= IotExtractType(monitor.Generator.ar_PhaseVoltage[2], 1, 1); 
// eDataMappingVarNames.Generator_ar_PhaseVoltage_L3: 				st_Variable:= IotExtractType(monitor.Generator.ar_PhaseVoltage[3], 1, 1); 
// eDataMappingVarNames.Generator_ar_Frequency_AVG: 				st_Variable:= IotExtractType(monitor.Generator.ar_Frequency[0], 2, 1); 
// eDataMappingVarNames.Generator_ar_Frequency_L1: 				st_Variable:= IotExtractType(monitor.Generator.ar_Frequency[1], 2, 1); 
// eDataMappingVarNames.Generator_ar_Frequency_L2: 				st_Variable:= IotExtractType(monitor.Generator.ar_Frequency[2], 2, 1); 
// eDataMappingVarNames.Generator_ar_Frequency_L3: 				st_Variable:= IotExtractType(monitor.Generator.ar_Frequency[3], 2, 1); 
// eDataMappingVarNames.Generator_ar_Current_AVG: 				st_Variable:= IotExtractType(monitor.Generator.ar_Current[0], 1, 1); 
// eDataMappingVarNames.Generator_ar_Current_L1: 				st_Variable:= IotExtractType(monitor.Generator.ar_Current[1], 1, 1); 
// eDataMappingVarNames.Generator_ar_Current_L2: 				st_Variable:= IotExtractType(monitor.Generator.ar_Current[2], 1, 1); 
// eDataMappingVarNames.Generator_ar_Current_L3: 				st_Variable:= IotExtractType(monitor.Generator.ar_Current[3], 1, 1); 
// eDataMappingVarNames.Generator_ar_PowerFactor_AVG: 				st_Variable:= IotExtractType(monitor.Generator.ar_PowerFactor[0], 2, 0); 
// eDataMappingVarNames.Generator_ar_ActivePower_AVG: 				st_Variable:= IotExtractType(monitor.Generator.ar_ActivePower[0], 1, 1); 
// eDataMappingVarNames.Generator_ar_ActivePower_L1: 				st_Variable:= IotExtractType(monitor.Generator.ar_ActivePower[1], 1, 1); 
// eDataMappingVarNames.Generator_ar_ActivePower_L2: 				st_Variable:= IotExtractType(monitor.Generator.ar_ActivePower[2], 1, 1); 
// eDataMappingVarNames.Generator_ar_ActivePower_L3: 				st_Variable:= IotExtractType(monitor.Generator.ar_ActivePower[3], 1, 1); 
// eDataMappingVarNames.Generator_ar_ReactivePower_AVG: 				st_Variable:= IotExtractType(monitor.Generator.ar_ReactivePower[0], 1, 1); 
// eDataMappingVarNames.Generator_ar_ApparentPower_AVG: 				st_Variable:= IotExtractType(monitor.Generator.ar_ApparentPower[0], 1, 1); 
// eDataMappingVarNames.HartingIO_b_DigitalInput1Active: 				st_Variable:= IotExtractType(monitor.HartingIO.b_DigitalInput1Active, 0, 0); 
// eDataMappingVarNames.HartingIO_b_DigitalInput2Active: 				st_Variable:= IotExtractType(monitor.HartingIO.b_DigitalInput2Active, 0, 0); 
// eDataMappingVarNames.HartingIO_b_GenLowFuel: 				st_Variable:= IotExtractType(monitor.HartingIO.b_GenLowFuel, 0, 0); 
// eDataMappingVarNames.HartingIO_b_ExtSystemShutdownRequest: 				st_Variable:= IotExtractType(monitor.HartingIO.b_ExtSystemShutdownRequest, 0, 0); 
// eDataMappingVarNames.HartingIO_b_ExtEMstopOK: 				st_Variable:= IotExtractType(monitor.HartingIO.b_ExtEMstopOK, 0, 0); 
// eDataMappingVarNames.HartingIO_b_ExtEMstopActive: 				st_Variable:= IotExtractType(monitor.HartingIO.b_ExtEMstopActive, 0, 0); 
END_CASE

IF index >= eDataMappingVarNames.controlfb_control_b_start AND index <= eDataMappingVarNames.controlfb_HardSettings_system_a_ui_OutputCurrentLimit_3 THEN
	st_RW.ReadFromNUC := aData[index].LogType <> 0;
	st_RW.WriteToNUC := FALSE;
ELSE
	st_RW.ReadFromNUC := FALSE;
	st_RW.WriteToNUC :=  aData[index].LogType <> 0;
END_IF


//-------------------------------Write to output---------------------------------------------
IotMappingV2.sName		:= aData[index].Label;				//Name of the variable
IotMappingV2.sValue		:= st_Variable.sValue;	//Extracted value of the variable
IotMappingV2.eUpdate	:= aData[index].LogInterval;				//Update frequency
IotMappingV2.st_RW		:= st_RW;				//Read/Write
IotMappingV2.pAdress	:= st_Variable.pAdress; //Adress pointer to variable
IotMappingV2.diSize		:= st_Variable.diSize;
IotMappingV2.ClassType	:= st_Variable.ClassType; //Extracted data type of the variable
IotMappingV2.bNumber	:= st_Variable.bNumber;
IotMappingV2.bJson		:= bJson;
END_METHOD

METHOD IoTWriteBacktoVar : BOOL;
VAR_INPUT
	sValue	  : STRING; //Content of variable to write to in STRING type
	pAdress	  : PVOID; //Adress of the Variable
	ClassType : __SYSTEM.TYPE_CLASS; //Type of the Variable
END_VAR

VAR
	pBool	: POINTER TO BOOL;
	pInt	: POINTER TO INT;
	pLreal	: POINTER TO LREAL;
	pWord	: POINTER TO WORD;
	pDword	: POINTER TO DWORD;
	pSint	: POINTER TO SINT;
	pReal	: POINTER TO REAL;
	pString : POINTER TO STRING;
END_VAR
CASE ClassType OF
    __SYSTEM.Type_Class.TYPE_BOOL :
		pBool:=pAdress;
		pBool^:=STRING_TO_BOOL(sValue);
    __SYSTEM.Type_Class.TYPE_ENUM :
		pInt:=pAdress;
		pInt^:=STRING_TO_INT(sValue);
    __SYSTEM.Type_Class.TYPE_LREAL :
		pLreal:=pAdress;
		pLreal^:=STRING_TO_LREAL(sValue);
    __SYSTEM.Type_Class.TYPE_WORD :
		pWord:=pAdress;
		pWord^:= STRING_TO_WORD(sValue);
    __SYSTEM.Type_Class.TYPE_DWORD :
		pDword:=pAdress;
		pDWord^:= STRING_TO_WORD(sValue);
    __SYSTEM.Type_Class.TYPE_SINT :
		pSint:=pAdress;
		pSint^:= STRING_TO_SINT(sValue);
    __SYSTEM.Type_Class.TYPE_INT :
		pInt:=pAdress;
		pInt^:=STRING_TO_INT(sValue);
    __SYSTEM.Type_Class.TYPE_REAL :
		pReal:=pAdress;
		pReal^:=STRING_TO_REAL(sValue);
    __SYSTEM.Type_Class.TYPE_STRING :	
		pString:=pAdress;
		pString^:=sValue;
		
	ELSE
		IoTWriteBackToVar:=FALSE;
END_CASE
END_METHOD

METHOD OrPublish : BOOL

VAR_INPUT
	iotprops 		: REFERENCE TO ST_IotProps;
	sOrPubPrefix	: STRING;
	sAssetID		: STRING;
END_VAR

VAR
	sTopic			: 	STRING;
	sQuote			:	STRING := '"';
END_VAR
//Prepare Topic		
sTopic:= concat(sORPubPrefix,IotProps.sName);
sTopic:= concat(sTopic,sAssetID);

//Catch NANs
IF IotProps.sValue = '#NaN' THEN
	IotProps.sValue:='0';
END_IF

//Convert payload to JSON string if text ( "sValue" )
IF NOT IotProps.bNumber AND NOT IotProps.bJson THEN
	concat2(ADR(sQuote), ADR(IotProps.sValue), ADR(IotProps.sValue), SIZEOF(IotProps.sValue));
	concat2(ADR(IotProps.sValue), ADR(sQuote), ADR(IotProps.sValue), SIZEOF(IotProps.sValue));
END_IF

//Publish 
fbMqttClient.Publish(sTopic:=sTopic,
pPayload := ADR(IotProps.sValue), //ADR(MessageToPublishJson),
nPayloadSize := LEN2(ADR(IotProps.sValue)), // ADR(MessageToPublishJson)),
eQoS := TcIotMqttQos.AtMostOnceDelivery,
bRetain:= FALSE,
bQueue := FALSE);
END_METHOD

METHOD PublishVarsV1 : BOOL
VAR_INPUT
END_VAR
b_UpdateActive := fbSendFastMessageTimer.Q OR fbSendSlowMessageTimer.Q OR bInitiateFirstTimeSend;
IF e_state = eConnectionState.authorized AND b_UpdateActive THEN
	FOR i:= 1 TO iSizeIotMappingV1 BY 1 DO	
			
		//----Get variable mapping properties corresponding to index
		st_IotProps:= IotMapping(i);
		
		//----Fast Message Sending
		IF (st_IotProps.eUpdate = eUpdate.Fast) AND st_IotProps.st_RW.WriteToNUC AND fbSendFastMessageTimer.Q THEN
				//Publish in OpenRemote format
				OrPublish(sOrPubPrefix:=sPubPrefix, sAssetID:=sAssetID, iotprops := st_IotProps);	
				//OrPublish(sOrPubPrefix:=sPubPrefix,sName:=st_IotProps.sName,sAssetID:=sAssetID,sValue:=st_IotProps.sValue, bNumber:=st_IotProps.bNumber);	
		END_IF
		
		//----Slow Message Sending---------
		IF (st_IotProps.eUpdate = eUpdate.Slow) AND st_IotProps.st_RW.WriteToNUC AND fbSendSlowMessageTimer.Q THEN		
				//Publish in OpenRemote format
				OrPublish(sOrPubPrefix:=sPubPrefix, sAssetID:=sAssetID, iotprops := st_IotProps);
		END_IF
		
		//----Maintenance Message Sending (sends every reconnect, which is reset daily)---------
		IF (st_IotProps.eUpdate = eUpdate.Daily) AND st_IotProps.st_RW.WriteToNUC AND bInitiateFirstTimeSend THEN		
				//Publish in OpenRemote format
				OrPublish(sOrPubPrefix:=sPubPrefix, sAssetID:=sAssetID, iotprops := st_IotProps);
		END_IF
		
		//----On change Message Sending------
		IF (st_IotProps.eUpdate = eUpdate.OnChange) AND st_IotProps.st_RW.WriteToNUC AND (fbSendFastMessageTimer.Q  OR bInitiateFirstTimeSend) THEN
			i_OnChangeValuesIndex := i_OnChangeValuesIndex + 1;
			
			//Evaluate whether value has changed or first time message trigger is active
			IF st_IotProps.sValue <> aPreviousValue[i_OnChangeValuesIndex] OR bInitiateFirstTimeSend THEN
				//Set current value to memory
				aPreviousValue[i_OnChangeValuesIndex]:= st_IotProps.sValue;
				//Publish in OpenRemote format
				OrPublish(sOrPubPrefix:=sPubPrefix, sAssetID:=sAssetID, iotprops := st_IotProps);

			END_IF
		END_IF	
	END_FOR
	i_OnChangeValuesIndex := 0;
	//Disable First Time send
	bInitiateFirstTimeSend:=FALSE;
END_IF
END_METHOD

METHOD PublishVarsV2 : BOOL
VAR_INPUT
	Authorized : BOOL;
	Interval : eUpdate;
END_VAR

VAR_IN_OUT
	state : ST_IOT_SentStateLog;
END_VAR

VAR
	Checksum : WORD;
	i : INT;
	Update : BOOL;
	CheckSumWordLast	: WORD;
END_VAR
IF Authorized AND State.bUpdate THEN
	State.bMessageSent := FALSE;
	FOR i:= State.LastIndexSent TO State.LastIndex BY 1 DO	
		//----Get variable mapping properties corresponding to index
//FIX MappingV2		//st_IotProps:= IotMappingV2(i);

		//---- Message Sending
		IF (st_IotProps.eUpdate = interval) AND st_IotProps.st_RW.WriteToNUC AND State.bUpdate THEN
			//Publish in OpenRemote format
			IF State.LastIndexSent < i THEN
				// onchange detection
				IF st_IotProps.eUpdate = eUpdate.OnChange THEN 
					CheckSum 	:= F_CheckSum16(st_IotProps.pAdress, st_iotProps.diSize, 0);
					Update := aCheckSumLast[i] <> CheckSum;
					aCheckSumLast[i] := CheckSum;
				ELSE
					Update := TRUE;
				END_IF
				
				//Update variable
				IF update THEN
					OrPublish(sOrPubPrefix:=sPubPrefix, sAssetID:=sAssetID, iotprops := st_IotProps);
					State.LastIndexSent := i;
					EXIT;
				END_IF
			END_IF
		END_IF
	END_FOR
ELSE
	RETURN;
END_IF

IF State.LastIndexSent = State.LastIndex AND State.bUpdate THEN
	State.bUpdate := FALSE;
	State.LastIndexSent := 0;
END_IF
END_METHOD

METHOD shutdown : BOOL
IF s_ShutdownFb = 'ERR' THEN
	w_shutdown := 0;
ELSE
	w_shutdown := 1;
END_IF

shutdown := s_ShutdownFb = 'OK';
END_METHOD

END_PROGRAM

(* stored: Version 1.1.0.1, ProductVersion 3.1.4026.18
   POU MqttComOpenremote: Id {892d67f6-1728-44e7-a46f-6c2166a8f218}, SpecialFunc None
   Method FillBatteryDatalog: Id {6de0f877-560b-463e-b91f-3c52ed293b96}
   Method IoTExtractType: Id {83d0dcf9-25e9-4193-b05f-dafb4eba6569}
   Method IotMapping: Id {a45dc000-ad50-4755-868e-776a573c193d}
   Method IoTMapping_json_X11: Id {a441caf9-2c7e-42fd-a5a2-e0203926b328}
   Method IoTMapping_json_X12: Id {7c59e038-b216-43a1-8872-8111b2c88571}
   Method IotMappingV2: Id {431eb580-3ed2-4a5c-8e42-394c707ae310}
   Method IoTWriteBacktoVar: Id {f5435517-1683-4bda-bc9b-0a22e1062dae}
   Method OrPublish: Id {5eeca784-63d0-471e-be07-c1f55dae6fe5}
   Method PublishVarsV1: Id {e7725402-5e07-4b2a-a16b-fafd3b1973f8}
   Method PublishVarsV2: Id {5cde2544-92ee-45d3-a3ae-1116f5b62fd4}
   Method shutdown: Id {b724972f-010b-4ca0-9b17-f3bb0308556a} *)
